LIN {X 0,Y 390.045,Z 635.903,A -85,B 0,C 180,E1 -11662.449,E2 -11662.449} C_VEL
LIN {X 0,Y 390.07,Z 635.897,A -85,B 0,C 180,E1 -11665.975,E2 -11665.975} C_VEL
LIN {X 0,Y 390.048,Z 635.899,A -85,B 0,C 180,E1 -11669.869,E2 -11669.869} C_VEL
LIN {X 0,Y 390.115,Z 635.892,A -85,B 0,C 180,E1 -11673.232,E2 -11673.232} C_VEL
LIN {X 0,Y 390.108,Z 635.894,A -85,B 0,C 180,E1 -11676.75,E2 -11676.75} C_VEL
LIN {X 0,Y 390.106,Z 635.893,A -85,B 0,C 180,E1 -11679.983,E2 -11679.983} C_VEL
LIN {X 0,Y 390.14,Z 635.89,A -85,B 0,C 180,E1 -11683.248,E2 -11683.248} C_VEL
LIN {X 0,Y 390.196,Z 635.883,A -85,B 0,C 180,E1 -11686.562,E2 -11686.562} C_VEL
LIN {X 0,Y 390.207,Z 635.88,A -85,B 0,C 180,E1 -11690.671,E2 -11690.671} C_VEL
LIN {X 0,Y 390.32,Z 635.867,A -85,B 0,C 180,E1 -11692.759,E2 -11692.759} C_VEL
LIN {X 0,Y 390.228,Z 635.88,A -85,B 0,C 180,E1 -11694.834,E2 -11694.834} C_VEL
LIN {X 0,Y 390.42,Z 635.855,A -85,B 0,C 180,E1 -11697.937,E2 -11697.937} C_VEL
LIN {X 0,Y 390.552,Z 635.838,A -85,B 0,C 180,E1 -11700,E2 -11700} C_VEL
LIN {X 0,Y 390.318,Z 635.869,A -85,B 0,C 180,E1 -11703.097,E2 -11703.097} C_VEL
LIN {X 0,Y 390.299,Z 635.869,A -85,B 0,C 180,E1 -11706.625,E2 -11706.625} C_VEL
LIN {X 0,Y 390.294,Z 635.871,A -85,B 0,C 180,E1 -11707.241,E2 -11707.241} C_VEL
LIN {X 0,Y 390.333,Z 637.799,A -85,B 0,C 180,E1 -11709.326,E2 -11709.326} C_VEL
LIN {X 0,Y 390.128,Z 641.266,A -85,B 0,C 180,E1 -11712.485,E2 -11712.485} C_VEL
LIN {X 0,Y 389.83,Z 644.908,A -85,B 0,C 180,E1 -11715.69,E2 -11715.69} C_VEL
LIN {X 0,Y 389.633,Z 648.746,A -85,B 0,C 180,E1 -11718.946,E2 -11718.946} C_VEL
LIN {X 0,Y 389.361,Z 652.799,A -85,B 0,C 180,E1 -11722.275,E2 -11722.275} C_VEL
LIN {X 0,Y 389.179,Z 657.06,A -85,B 0,C 180,E1 -11725.684,E2 -11725.684} C_VEL
LIN {X 0,Y 389.178,Z 658.085,A -85,B 0,C 180,E1 -11726.332,E2 -11726.332} C_VEL
LIN {X 0,Y 392.474,Z 670.829,A -85,B 0,C 180,E1 -11726.99,E2 -11726.99} C_VEL
LIN {X 0,Y 394.705,Z 682.309,A -85,B 0,C 180,E1 -11727.722,E2 -11727.722} C_VEL
LIN {X 0,Y 394.988,Z 685.201,A -85,B 0,C 180,E1 -11727.916,E2 -11727.916} C_VEL
LIN {X 0,Y 394.073,Z 697.293,A -85,B 0,C 180,E1 -11728.785,E2 -11728.785} C_VEL
LIN {X 0,Y 393.149,Z 709.316,A -85,B 0,C 180,E1 -11729.905,E2 -11729.905} C_VEL
LIN {X 0,Y 392.133,Z 719.9,A -85,B 0,C 180,E1 -11731.156,E2 -11731.156} C_VEL
LIN {X 0,Y 391.275,Z 729.716,A -85,B 0,C 180,E1 -11732.606,E2 -11732.606} C_VEL
LIN {X 0,Y 390.488,Z 737.933,A -85,B 0,C 180,E1 -11734.115,E2 -11734.115} C_VEL
LIN {X 0,Y 389.802,Z 745.117,A -85,B 0,C 180,E1 -11735.773,E2 -11735.773} C_VEL
LIN {X 0,Y 389.344,Z 750.732,A -85,B 0,C 180,E1 -11737.416,E2 -11737.416} C_VEL
LIN {X 0,Y 389,Z 755.433,A -85,B 0,C 180,E1 -11739.223,E2 -11739.223} C_VEL
LIN {X 0,Y 388.797,Z 758.049,A -85,B 0,C 180,E1 -11740.606,E2 -11740.606} C_VEL
LIN {X 0,Y 388.642,Z 760.083,A -85,B 0,C 180,E1 -11742.147,E2 -11742.147} C_VEL
LIN {X 0,Y 388.547,Z 761.204,A -85,B 0,C 180,E1 -11743.654,E2 -11743.654} C_VEL
LIN {X 0,Y 388.507,Z 761.496,A -85,B 0,C 180,E1 -11745.13,E2 -11745.13} C_VEL
LIN {X 0,Y 388.52,Z 761.002,A -85,B 0,C 180,E1 -11746.576,E2 -11746.576} C_VEL
LIN {X 0,Y 388.613,Z 759.717,A -85,B 0,C 180,E1 -11747.999,E2 -11747.999} C_VEL
LIN {X 0,Y 388.87,Z 756.445,A -85,B 0,C 180,E1 -11750.089,E2 -11750.089} C_VEL
LIN {X 0,Y 389.073,Z 753.106,A -85,B 0,C 180,E1 -11751.549,E2 -11751.549} C_VEL
LIN {X 0,Y 389.47,Z 747.243,A -85,B 0,C 180,E1 -11753.452,E2 -11753.452} C_VEL
LIN {X 0,Y 390.007,Z 740.747,A -85,B 0,C 180,E1 -11755.082,E2 -11755.082} C_VEL
LIN {X 0,Y 390.537,Z 734.245,A -85,B 0,C 180,E1 -11756.401,E2 -11756.401} C_VEL
LIN {X 0,Y 391.291,Z 725.804,A -85,B 0,C 180,E1 -11757.81,E2 -11757.81} C_VEL
LIN {X 0,Y 392.183,Z 715.296,A -85,B 0,C 180,E1 -11759.218,E2 -11759.218} C_VEL
LIN {X 0,Y 393.07,Z 704.453,A -85,B 0,C 180,E1 -11760.382,E2 -11760.382} C_VEL
LIN {X 0,Y 393.86,Z 693.01,A -85,B 0,C 180,E1 -11761.351,E2 -11761.351} C_VEL
LIN {X 0,Y 394.476,Z 683.755,A -85,B 0,C 180,E1 -11761.977,E2 -11761.977} C_VEL
LIN {X 0,Y 392.239,Z 671.38,A -85,B 0,C 180,E1 -11762.74,E2 -11762.74} C_VEL
LIN {X 0,Y 389.29,Z 658.629,A -85,B 0,C 180,E1 -11763.351,E2 -11763.351} C_VEL
LIN {X 0,Y 389.019,Z 657.042,A -85,B 0,C 180,E1 -11763.44,E2 -11763.44} C_VEL
LIN {X 0,Y 389.155,Z 652.247,A -85,B 0,C 180,E1 -11767.08,E2 -11767.08} C_VEL
LIN {X 0,Y 389.385,Z 648.528,A -85,B 0,C 180,E1 -11769.944,E2 -11769.944} C_VEL
LIN {X 0,Y 389.561,Z 644.36,A -85,B 0,C 180,E1 -11773.222,E2 -11773.222} C_VEL
LIN {X 0,Y 389.876,Z 639.95,A -85,B 0,C 180,E1 -11776.76,E2 -11776.76} C_VEL
LIN {X 0,Y 389.963,Z 636.512,A -85,B 0,C 180,E1 -11779.617,E2 -11779.617} C_VEL
LIN {X 0,Y 390.071,Z 635.898,A -85,B 0,C 180,E1 -11780.668,E2 -11780.668} C_VEL
LIN {X 0,Y 390.293,Z 635.871,A -85,B 0,C 180,E1 -11782.758,E2 -11782.758} C_VEL
LIN {X 0,Y 390.229,Z 635.879,A -85,B 0,C 180,E1 -11784.833,E2 -11784.833} C_VEL
LIN {X 0,Y 390.424,Z 635.849,A -85,B 0,C 180,E1 -11787.936,E2 -11787.936} C_VEL
LIN {X 0,Y 390.554,Z 635.834,A -85,B 0,C 180,E1 -11790,E2 -11790} C_VEL
LIN {X 0,Y 390.318,Z 635.867,A -85,B 0,C 180,E1 -11793.096,E2 -11793.096} C_VEL
LIN {X 0,Y 390.313,Z 635.864,A -85,B 0,C 180,E1 -11796.202,E2 -11796.202} C_VEL
LIN {X 0,Y 390.171,Z 635.883,A -85,B 0,C 180,E1 -11798.285,E2 -11798.285} C_VEL
LIN {X 0,Y 389.679,Z 635.945,A -85,B 0,C 180,E1 -11801.442,E2 -11801.442} C_VEL
LIN {X 0,Y 389.557,Z 636.18,A -85,B 0,C 180,E1 -11802.238,E2 -11802.238} C_VEL
LIN {X 0,Y 389.338,Z 640.085,A -85,B 0,C 180,E1 -11804.837,E2 -11804.837} C_VEL
LIN {X 0,Y 388.609,Z 641.43,A -85,B 0,C 180,E1 -11805.677,E2 -11805.677} C_VEL
LIN {X 0,Y 385.67,Z 643.774,A -85,B 0,C 180,E1 -11807.034,E2 -11807.034} C_VEL
LIN {X 0,Y 383.212,Z 645.663,A -85,B 0,C 180,E1 -11808.131,E2 -11808.131} C_VEL
LIN {X 0,Y 382.164,Z 647.033,A -85,B 0,C 180,E1 -11808.983,E2 -11808.983} C_VEL
LIN {X 0,Y 382.081,Z 647.468,A -85,B 0,C 180,E1 -11809.272,E2 -11809.272} C_VEL
LIN {X 0,Y 381.91,Z 653.113,A -85,B 0,C 180,E1 -11813.057,E2 -11813.057} C_VEL
LIN {X 0,Y 381.878,Z 656.667,A -85,B 0,C 180,E1 -11815.387,E2 -11815.387} C_VEL
LIN {X 0,Y 384.96,Z 670.347,A -85,B 0,C 180,E1 -11816.022,E2 -11816.022} C_VEL
LIN {X 0,Y 387.385,Z 683.195,A -85,B 0,C 180,E1 -11816.826,E2 -11816.826} C_VEL
LIN {X 0,Y 386.877,Z 694.197,A -85,B 0,C 180,E1 -11817.595,E2 -11817.595} C_VEL
LIN {X 0,Y 385.998,Z 705.968,A -85,B 0,C 180,E1 -11818.634,E2 -11818.634} C_VEL
LIN {X 0,Y 385.071,Z 716.555,A -85,B 0,C 180,E1 -11819.824,E2 -11819.824} C_VEL
LIN {X 0,Y 384.168,Z 726.914,A -85,B 0,C 180,E1 -11821.271,E2 -11821.271} C_VEL
LIN {X 0,Y 383.482,Z 734.296,A -85,B 0,C 180,E1 -11822.538,E2 -11822.538} C_VEL
LIN {X 0,Y 382.975,Z 740.583,A -85,B 0,C 180,E1 -11823.836,E2 -11823.836} C_VEL
LIN {X 0,Y 382.455,Z 746.653,A -85,B 0,C 180,E1 -11825.356,E2 -11825.356} C_VEL
LIN {X 0,Y 382.09,Z 751.026,A -85,B 0,C 180,E1 -11826.711,E2 -11826.711} C_VEL
LIN {X 0,Y 381.844,Z 754.811,A -85,B 0,C 180,E1 -11828.181,E2 -11828.181} C_VEL
LIN {X 0,Y 381.522,Z 758.493,A -85,B 0,C 180,E1 -11830.145,E2 -11830.145} C_VEL
LIN {X 0,Y 381.417,Z 760.21,A -85,B 0,C 180,E1 -11831.554,E2 -11831.554} C_VEL
LIN {X 0,Y 381.35,Z 761.195,A -85,B 0,C 180,E1 -11832.99,E2 -11832.99} C_VEL
LIN {X 0,Y 381.403,Z 761.452,A -85,B 0,C 180,E1 -11834.443,E2 -11834.443} C_VEL
LIN {X 0,Y 381.435,Z 760.939,A -85,B 0,C 180,E1 -11835.936,E2 -11835.936} C_VEL
LIN {X 0,Y 381.547,Z 759.581,A -85,B 0,C 180,E1 -11837.458,E2 -11837.458} C_VEL
LIN {X 0,Y 381.702,Z 757.288,A -85,B 0,C 180,E1 -11839.016,E2 -11839.016} C_VEL
LIN {X 0,Y 382.005,Z 753.991,A -85,B 0,C 180,E1 -11840.596,E2 -11840.596} C_VEL
LIN {X 0,Y 382.384,Z 749.518,A -85,B 0,C 180,E1 -11842.214,E2 -11842.214} C_VEL
LIN {X 0,Y 382.967,Z 742.914,A -85,B 0,C 180,E1 -11844.038,E2 -11844.038} C_VEL
LIN {X 0,Y 383.596,Z 736.113,A -85,B 0,C 180,E1 -11845.533,E2 -11845.533} C_VEL
LIN {X 0,Y 384.492,Z 727.815,A -85,B 0,C 180,E1 -11847.013,E2 -11847.013} C_VEL
LIN {X 0,Y 385.344,Z 719.065,A -85,B 0,C 180,E1 -11848.285,E2 -11848.285} C_VEL
LIN {X 0,Y 386.37,Z 708.31,A -85,B 0,C 180,E1 -11849.548,E2 -11849.548} C_VEL
LIN {X 0,Y 387.261,Z 697.305,A -85,B 0,C 180,E1 -11850.586,E2 -11850.586} C_VEL
LIN {X 0,Y 388.115,Z 685.408,A -85,B 0,C 180,E1 -11851.453,E2 -11851.453} C_VEL
LIN {X 0,Y 386.153,Z 673.731,A -85,B 0,C 180,E1 -11852.242,E2 -11852.242} C_VEL
LIN {X 0,Y 383.142,Z 661.505,A -85,B 0,C 180,E1 -11852.926,E2 -11852.926} C_VEL
LIN {X 0,Y 381.987,Z 657.119,A -85,B 0,C 180,E1 -11853.133,E2 -11853.133} C_VEL
LIN {X 0,Y 382.071,Z 652.636,A -85,B 0,C 180,E1 -11856.129,E2 -11856.129} C_VEL
LIN {X 0,Y 382.223,Z 647.235,A -85,B 0,C 180,E1 -11859.674,E2 -11859.674} C_VEL
LIN {X 0,Y 382.36,Z 642.32,A -85,B 0,C 180,E1 -11862.897,E2 -11862.897} C_VEL
LIN {X 0,Y 382.677,Z 636.826,A -85,B 0,C 180,E1 -11866.478,E2 -11866.478} C_VEL
LIN {X 0,Y 383.006,Z 636.779,A -85,B 0,C 180,E1 -11869.426,E2 -11869.426} C_VEL
LIN {X 0,Y 383.25,Z 636.75,A -85,B 0,C 180,E1 -11872.625,E2 -11872.625} C_VEL
LIN {X 0,Y 383.196,Z 636.756,A -85,B 0,C 180,E1 -11874.738,E2 -11874.738} C_VEL
LIN {X 0,Y 383.385,Z 636.731,A -85,B 0,C 180,E1 -11877.899,E2 -11877.899} C_VEL
LIN {X 0,Y 383.518,Z 636.715,A -85,B 0,C 180,E1 -11880,E2 -11880} C_VEL
LIN {X 0,Y 383.249,Z 636.749,A -85,B 0,C 180,E1 -11883.154,E2 -11883.154} C_VEL
LIN {X 0,Y 383.284,Z 636.743,A -85,B 0,C 180,E1 -11886.316,E2 -11886.316} C_VEL
LIN {X 0,Y 383.256,Z 636.747,A -85,B 0,C 180,E1 -11888.436,E2 -11888.436} C_VEL
LIN {X 0,Y 383.095,Z 636.766,A -85,B 0,C 180,E1 -11891.642,E2 -11891.642} C_VEL
LIN {X 0,Y 383.106,Z 636.766,A -85,B 0,C 180,E1 -11894.882,E2 -11894.882} C_VEL
LIN {X 0,Y 383.085,Z 636.768,A -85,B 0,C 180,E1 -11898.172,E2 -11898.172} C_VEL
LIN {X 0,Y 382.989,Z 636.777,A -85,B 0,C 180,E1 -11901.531,E2 -11901.531} C_VEL
LIN {X 0,Y 383.049,Z 636.773,A -85,B 0,C 180,E1 -11904.961,E2 -11904.961} C_VEL
LIN {X 0,Y 383.046,Z 636.77,A -85,B 0,C 180,E1 -11908.492,E2 -11908.492} C_VEL
LIN {X 0,Y 383.008,Z 636.779,A -85,B 0,C 180,E1 -11912.15,E2 -11912.15} C_VEL
LIN {X 0,Y 383.015,Z 636.776,A -85,B 0,C 180,E1 -11914.668,E2 -11914.668} C_VEL
LIN {X 0,Y 382.999,Z 636.777,A -85,B 0,C 180,E1 -11917.905,E2 -11917.905} C_VEL
LIN {X 0,Y 382.981,Z 636.781,A -85,B 0,C 180,E1 -11921.348,E2 -11921.348} C_VEL
LIN {X 0,Y 382.993,Z 636.78,A -85,B 0,C 180,E1 -11924.304,E2 -11924.304} C_VEL
LIN {X 0,Y 383.029,Z 636.776,A -85,B 0,C 180,E1 -11928.132,E2 -11928.132} C_VEL
LIN {X 0,Y 383.63,Z 640,A -85,B 0,C 180,E1 -11930.303,E2 -11930.303} C_VEL
LIN {X 0,Y 384.197,Z 644.117,A -85,B 0,C 180,E1 -11932.868,E2 -11932.868} C_VEL
LIN {X 0,Y 384.255,Z 648.497,A -85,B 0,C 180,E1 -11935.46,E2 -11935.46} C_VEL
LIN {X 0,Y 383.782,Z 653.949,A -85,B 0,C 180,E1 -11938.541,E2 -11938.541} C_VEL
LIN {X 0,Y 383.349,Z 659.601,A -85,B 0,C 180,E1 -11941.642,E2 -11941.642} C_VEL
LIN {X 0,Y 382.888,Z 665.937,A -85,B 0,C 180,E1 -11945.029,E2 -11945.029} C_VEL
LIN {X 0,Y 382.537,Z 672.453,A -85,B 0,C 180,E1 -11948.443,E2 -11948.443} C_VEL
LIN {X 0,Y 382.233,Z 677.92,A -85,B 0,C 180,E1 -11951.214,E2 -11951.214} C_VEL
LIN {X 0,Y 384.658,Z 691.057,A -85,B 0,C 180,E1 -11951.82,E2 -11951.82} C_VEL
LIN {X 0,Y 386.51,Z 704.837,A -85,B 0,C 180,E1 -11952.638,E2 -11952.638} C_VEL
LIN {X 0,Y 387.056,Z 710.39,A -85,B 0,C 180,E1 -11953.022,E2 -11953.022} C_VEL
LIN {X 0,Y 386.176,Z 721.714,A -85,B 0,C 180,E1 -11953.887,E2 -11953.887} C_VEL
LIN {X 0,Y 385.325,Z 732.5,A -85,B 0,C 180,E1 -11954.936,E2 -11954.936} C_VEL
LIN {X 0,Y 384.394,Z 743.32,A -85,B 0,C 180,E1 -11956.251,E2 -11956.251} C_VEL
LIN {X 0,Y 383.627,Z 752.108,A -85,B 0,C 180,E1 -11957.57,E2 -11957.57} C_VEL
LIN {X 0,Y 382.854,Z 760.667,A -85,B 0,C 180,E1 -11959.155,E2 -11959.155} C_VEL
LIN {X 0,Y 382.309,Z 767.528,A -85,B 0,C 180,E1 -11960.744,E2 -11960.744} C_VEL
LIN {X 0,Y 381.868,Z 773.826,A -85,B 0,C 180,E1 -11962.599,E2 -11962.599} C_VEL
LIN {X 0,Y 381.697,Z 777.168,A -85,B 0,C 180,E1 -11963.868,E2 -11963.868} C_VEL
LIN {X 0,Y 381.633,Z 780.953,A -85,B 0,C 180,E1 -11965.776,E2 -11965.776} C_VEL
LIN {X 0,Y 381.545,Z 782.431,A -85,B 0,C 180,E1 -11966.833,E2 -11966.833} C_VEL
LIN {X 0,Y 381.616,Z 784.105,A -85,B 0,C 180,E1 -11968.945,E2 -11968.945} C_VEL
LIN {X 0,Y 381.639,Z 784.353,A -85,B 0,C 180,E1 -11970,E2 -11970} C_VEL
LIN {X 0,Y 381.616,Z 784.185,A -85,B 0,C 180,E1 -11971.056,E2 -11971.056} C_VEL
LIN {X 0,Y 381.544,Z 782.599,A -85,B 0,C 180,E1 -11973.168,E2 -11973.168} C_VEL
LIN {X 0,Y 381.634,Z 781.213,A -85,B 0,C 180,E1 -11974.225,E2 -11974.225} C_VEL
LIN {X 0,Y 381.734,Z 777.457,A -85,B 0,C 180,E1 -11976.184,E2 -11976.184} C_VEL
LIN {X 0,Y 382.012,Z 772.753,A -85,B 0,C 180,E1 -11977.931,E2 -11977.931} C_VEL
LIN {X 0,Y 382.498,Z 766.218,A -85,B 0,C 180,E1 -11979.786,E2 -11979.786} C_VEL
LIN {X 0,Y 383.092,Z 759.074,A -85,B 0,C 180,E1 -11981.374,E2 -11981.374} C_VEL
LIN {X 0,Y 384.032,Z 750.186,A -85,B 0,C 180,E1 -11982.955,E2 -11982.955} C_VEL
LIN {X 0,Y 384.832,Z 740.922,A -85,B 0,C 180,E1 -11984.299,E2 -11984.299} C_VEL
LIN {X 0,Y 385.707,Z 731.154,A -85,B 0,C 180,E1 -11985.455,E2 -11985.455} C_VEL
LIN {X 0,Y 386.704,Z 720.176,A -85,B 0,C 180,E1 -11986.498,E2 -11986.498} C_VEL
LIN {X 0,Y 387.423,Z 709.101,A -85,B 0,C 180,E1 -11987.34,E2 -11987.34} C_VEL
LIN {X 0,Y 386.021,Z 696.528,A -85,B 0,C 180,E1 -11988.181,E2 -11988.181} C_VEL
LIN {X 0,Y 383.884,Z 684.526,A -85,B 0,C 180,E1 -11988.827,E2 -11988.827} C_VEL
LIN {X 0,Y 382.267,Z 677.169,A -85,B 0,C 180,E1 -11989.162,E2 -11989.162} C_VEL
LIN {X 0,Y 382.62,Z 671.462,A -85,B 0,C 180,E1 -11992.12,E2 -11992.12} C_VEL
LIN {X 0,Y 383.018,Z 664.285,A -85,B 0,C 180,E1 -11995.959,E2 -11995.959} C_VEL
LIN {X 0,Y 383.468,Z 658.701,A -85,B 0,C 180,E1 -11999.057,E2 -11999.057} C_VEL
LIN {X 0,Y 384.047,Z 652.474,A -85,B 0,C 180,E1 -12002.67,E2 -12002.67} C_VEL
LIN {X 0,Y 384.393,Z 649.227,A -85,B 0,C 180,E1 -12004.639,E2 -12004.639} C_VEL
LIN {X 0,Y 384.313,Z 645.402,A -85,B 0,C 180,E1 -12007.12,E2 -12007.12} C_VEL
LIN {X 0,Y 383.808,Z 641.495,A -85,B 0,C 180,E1 -12009.859,E2 -12009.859} C_VEL
LIN {X 0,Y 383.035,Z 636.776,A -85,B 0,C 180,E1 -12013.567,E2 -12013.567} C_VEL
LIN {X 0,Y 383.012,Z 636.78,A -85,B 0,C 180,E1 -12017.24,E2 -12017.24} C_VEL
LIN {X 0,Y 383.017,Z 636.778,A -85,B 0,C 180,E1 -12020.414,E2 -12020.414} C_VEL
LIN {X 0,Y 383.027,Z 636.776,A -85,B 0,C 180,E1 -12024.045,E2 -12024.045} C_VEL
LIN {X 0,Y 382.988,Z 636.779,A -85,B 0,C 180,E1 -12027.578,E2 -12027.578} C_VEL
LIN {X 0,Y 382.994,Z 636.779,A -85,B 0,C 180,E1 -12030.3,E2 -12030.3} C_VEL
LIN {X 0,Y 383.082,Z 636.766,A -85,B 0,C 180,E1 -12034.021,E2 -12034.021} C_VEL
LIN {X 0,Y 383.01,Z 636.778,A -85,B 0,C 180,E1 -12037.335,E2 -12037.335} C_VEL
LIN {X 0,Y 383.062,Z 636.772,A -85,B 0,C 180,E1 -12040.716,E2 -12040.716} C_VEL
LIN {X 0,Y 383.082,Z 636.768,A -85,B 0,C 180,E1 -12044.027,E2 -12044.027} C_VEL
LIN {X 0,Y 383.138,Z 636.761,A -85,B 0,C 180,E1 -12047.284,E2 -12047.284} C_VEL
LIN {X 0,Y 383.153,Z 636.758,A -85,B 0,C 180,E1 -12050.498,E2 -12050.498} C_VEL
LIN {X 0,Y 383.275,Z 636.743,A -85,B 0,C 180,E1 -12052.625,E2 -12052.625} C_VEL
LIN {X 0,Y 383.201,Z 636.754,A -85,B 0,C 180,E1 -12054.739,E2 -12054.739} C_VEL
LIN {X 0,Y 383.387,Z 636.731,A -85,B 0,C 180,E1 -12057.899,E2 -12057.899} C_VEL
LIN {X 0,Y 383.521,Z 636.714,A -85,B 0,C 180,E1 -12060,E2 -12060} C_VEL
LIN {X 0,Y 383.254,Z 636.75,A -85,B 0,C 180,E1 -12063.154,E2 -12063.154} C_VEL
LIN {X 0,Y 383.271,Z 636.803,A -85,B 0,C 180,E1 -12066.622,E2 -12066.622} C_VEL
LIN {X 0,Y 383.287,Z 636.949,A -85,B 0,C 180,E1 -12067.374,E2 -12067.374} C_VEL
LIN {X 0,Y 383.241,Z 640.208,A -85,B 0,C 180,E1 -12070.567,E2 -12070.567} C_VEL
LIN {X 0,Y 382.991,Z 643.756,A -85,B 0,C 180,E1 -12073.801,E2 -12073.801} C_VEL
LIN {X 0,Y 382.689,Z 647.682,A -85,B 0,C 180,E1 -12077.26,E2 -12077.26} C_VEL
LIN {X 0,Y 382.449,Z 651.413,A -85,B 0,C 180,E1 -12080.435,E2 -12080.435} C_VEL
LIN {X 0,Y 382.211,Z 655.568,A -85,B 0,C 180,E1 -12083.862,E2 -12083.862} C_VEL
LIN {X 0,Y 382.103,Z 658.125,A -85,B 0,C 180,E1 -12085.928,E2 -12085.928} C_VEL
LIN {X 0,Y 385.596,Z 671.291,A -85,B 0,C 180,E1 -12086.631,E2 -12086.631} C_VEL
LIN {X 0,Y 387.809,Z 682.676,A -85,B 0,C 180,E1 -12087.377,E2 -12087.377} C_VEL
LIN {X 0,Y 388.111,Z 687.57,A -85,B 0,C 180,E1 -12087.72,E2 -12087.72} C_VEL
LIN {X 0,Y 387.174,Z 699.209,A -85,B 0,C 180,E1 -12088.605,E2 -12088.605} C_VEL
LIN {X 0,Y 386.243,Z 710.637,A -85,B 0,C 180,E1 -12089.725,E2 -12089.725} C_VEL
LIN {X 0,Y 385.225,Z 720.768,A -85,B 0,C 180,E1 -12090.967,E2 -12090.967} C_VEL
LIN {X 0,Y 384.345,Z 729.91,A -85,B 0,C 180,E1 -12092.35,E2 -12092.35} C_VEL
LIN {X 0,Y 383.538,Z 737.997,A -85,B 0,C 180,E1 -12093.858,E2 -12093.858} C_VEL
LIN {X 0,Y 382.779,Z 745.636,A -85,B 0,C 180,E1 -12095.658,E2 -12095.658} C_VEL
LIN {X 0,Y 382.277,Z 751.252,A -85,B 0,C 180,E1 -12097.351,E2 -12097.351} C_VEL
LIN {X 0,Y 381.998,Z 754.801,A -85,B 0,C 180,E1 -12098.721,E2 -12098.721} C_VEL
LIN {X 0,Y 381.785,Z 757.62,A -85,B 0,C 180,E1 -12100.113,E2 -12100.113} C_VEL
LIN {X 0,Y 381.582,Z 759.732,A -85,B 0,C 180,E1 -12101.533,E2 -12101.533} C_VEL
LIN {X 0,Y 381.502,Z 761.063,A -85,B 0,C 180,E1 -12102.97,E2 -12102.97} C_VEL
LIN {X 0,Y 381.421,Z 761.675,A -85,B 0,C 180,E1 -12104.442,E2 -12104.442} C_VEL
LIN {X 0,Y 381.412,Z 761.516,A -85,B 0,C 180,E1 -12105.941,E2 -12105.941} C_VEL
LIN {X 0,Y 381.468,Z 760.524,A -85,B 0,C 180,E1 -12107.472,E2 -12107.472} C_VEL
LIN {X 0,Y 381.637,Z 758.614,A -85,B 0,C 180,E1 -12109.029,E2 -12109.029} C_VEL
LIN {X 0,Y 381.853,Z 755.698,A -85,B 0,C 180,E1 -12110.625,E2 -12110.625} C_VEL
LIN {X 0,Y 382.095,Z 751.605,A -85,B 0,C 180,E1 -12112.271,E2 -12112.271} C_VEL
LIN {X 0,Y 382.574,Z 745.965,A -85,B 0,C 180,E1 -12113.995,E2 -12113.995} C_VEL
LIN {X 0,Y 383.121,Z 739.116,A -85,B 0,C 180,E1 -12115.638,E2 -12115.638} C_VEL
LIN {X 0,Y 383.792,Z 731.872,A -85,B 0,C 180,E1 -12117.045,E2 -12117.045} C_VEL
LIN {X 0,Y 384.653,Z 722.225,A -85,B 0,C 180,E1 -12118.57,E2 -12118.57} C_VEL
LIN {X 0,Y 385.647,Z 711.389,A -85,B 0,C 180,E1 -12119.923,E2 -12119.923} C_VEL
LIN {X 0,Y 386.502,Z 700.447,A -85,B 0,C 180,E1 -12121.02,E2 -12121.02} C_VEL
LIN {X 0,Y 387.303,Z 689.022,A -85,B 0,C 180,E1 -12121.922,E2 -12121.922} C_VEL
LIN {X 0,Y 387.451,Z 683.305,A -85,B 0,C 180,E1 -12122.302,E2 -12122.302} C_VEL
LIN {X 0,Y 384.754,Z 669.527,A -85,B 0,C 180,E1 -12123.159,E2 -12123.159} C_VEL
LIN {X 0,Y 382.003,Z 657.244,A -85,B 0,C 180,E1 -12123.76,E2 -12123.76} C_VEL
LIN {X 0,Y 382.105,Z 652.674,A -85,B 0,C 180,E1 -12127.278,E2 -12127.278} C_VEL
LIN {X 0,Y 382.332,Z 648.341,A -85,B 0,C 180,E1 -12130.678,E2 -12130.678} C_VEL
LIN {X 0,Y 382.533,Z 644.196,A -85,B 0,C 180,E1 -12134.003,E2 -12134.003} C_VEL
LIN {X 0,Y 382.858,Z 640.183,A -85,B 0,C 180,E1 -12137.274,E2 -12137.274} C_VEL
LIN {X 0,Y 382.895,Z 637.635,A -85,B 0,C 180,E1 -12139.423,E2 -12139.423} C_VEL
LIN {X 0,Y 382.996,Z 636.779,A -85,B 0,C 180,E1 -12140.494,E2 -12140.494} C_VEL
LIN {X 0,Y 383.242,Z 636.747,A -85,B 0,C 180,E1 -12142.624,E2 -12142.624} C_VEL
LIN {X 0,Y 383.201,Z 636.754,A -85,B 0,C 180,E1 -12144.738,E2 -12144.738} C_VEL
LIN {X 0,Y 383.391,Z 636.725,A -85,B 0,C 180,E1 -12147.899,E2 -12147.899} C_VEL
LIN {X 0,Y 383.523,Z 636.709,A -85,B 0,C 180,E1 -12150,E2 -12150} C_VEL
LIN {X 0,Y 383.254,Z 636.746,A -85,B 0,C 180,E1 -12153.153,E2 -12153.153} C_VEL
LIN {X 0,Y 383.265,Z 636.743,A -85,B 0,C 180,E1 -12156.316,E2 -12156.316} C_VEL
LIN {X 0,Y 383.106,Z 636.764,A -85,B 0,C 180,E1 -12158.439,E2 -12158.439} C_VEL
LIN {X 0,Y 382.547,Z 636.833,A -85,B 0,C 180,E1 -12162.096,E2 -12162.096} C_VEL
LIN {X 0,Y 382.258,Z 642.612,A -85,B 0,C 180,E1 -12166.008,E2 -12166.008} C_VEL
LIN {X 0,Y 382.081,Z 647.468,A -85,B 0,C 180,E1 -12169.272,E2 -12169.272} C_VEL
LIN {X 0,Y 381.403,Z 648.808,A -85,B 0,C 180,E1 -12170.128,E2 -12170.128} C_VEL
LIN {X 0,Y 378.476,Z 651.152,A -85,B 0,C 180,E1 -12171.512,E2 -12171.512} C_VEL
LIN {X 0,Y 375.98,Z 653.04,A -85,B 0,C 180,E1 -12172.63,E2 -12172.63} C_VEL
LIN {X 0,Y 374.892,Z 654.419,A -85,B 0,C 180,E1 -12173.498,E2 -12173.498} C_VEL
LIN {X 0,Y 374.795,Z 654.862,A -85,B 0,C 180,E1 -12173.793,E2 -12173.793} C_VEL
LIN {X 0,Y 374.785,Z 656.69,A -85,B 0,C 180,E1 -12175.029,E2 -12175.029} C_VEL
LIN {X 0,Y 378.148,Z 671.675,A -85,B 0,C 180,E1 -12175.772,E2 -12175.772} C_VEL
LIN {X 0,Y 380.536,Z 684.409,A -85,B 0,C 180,E1 -12176.606,E2 -12176.606} C_VEL
LIN {X 0,Y 379.958,Z 695.309,A -85,B 0,C 180,E1 -12177.396,E2 -12177.396} C_VEL
LIN {X 0,Y 379.119,Z 705.958,A -85,B 0,C 180,E1 -12178.361,E2 -12178.361} C_VEL
LIN {X 0,Y 378.204,Z 716.023,A -85,B 0,C 180,E1 -12179.498,E2 -12179.498} C_VEL
LIN {X 0,Y 377.388,Z 725.09,A -85,B 0,C 180,E1 -12180.755,E2 -12180.755} C_VEL
LIN {X 0,Y 376.612,Z 733.265,A -85,B 0,C 180,E1 -12182.129,E2 -12182.129} C_VEL
LIN {X 0,Y 375.907,Z 741.288,A -85,B 0,C 180,E1 -12183.793,E2 -12183.793} C_VEL
LIN {X 0,Y 375.345,Z 747.708,A -85,B 0,C 180,E1 -12185.481,E2 -12185.481} C_VEL
LIN {X 0,Y 374.849,Z 753.478,A -85,B 0,C 180,E1 -12187.445,E2 -12187.445} C_VEL
LIN {X 0,Y 374.604,Z 756.736,A -85,B 0,C 180,E1 -12188.938,E2 -12188.938} C_VEL
LIN {X 0,Y 374.353,Z 759.926,A -85,B 0,C 180,E1 -12191.077,E2 -12191.077} C_VEL
LIN {X 0,Y 374.252,Z 761.354,A -85,B 0,C 180,E1 -12192.914,E2 -12192.914} C_VEL
LIN {X 0,Y 374.306,Z 761.65,A -85,B 0,C 180,E1 -12194.48,E2 -12194.48} C_VEL
LIN {X 0,Y 374.341,Z 761.137,A -85,B 0,C 180,E1 -12196,E2 -12196} C_VEL
LIN {X 0,Y 374.455,Z 759.84,A -85,B 0,C 180,E1 -12197.494,E2 -12197.494} C_VEL
LIN {X 0,Y 374.612,Z 757.777,A -85,B 0,C 180,E1 -12198.957,E2 -12198.957} C_VEL
LIN {X 0,Y 374.879,Z 754.965,A -85,B 0,C 180,E1 -12200.401,E2 -12200.401} C_VEL
LIN {X 0,Y 375.298,Z 750.255,A -85,B 0,C 180,E1 -12202.21,E2 -12202.21} C_VEL
LIN {X 0,Y 375.694,Z 745.808,A -85,B 0,C 180,E1 -12203.55,E2 -12203.55} C_VEL
LIN {X 0,Y 376.409,Z 738.896,A -85,B 0,C 180,E1 -12205.237,E2 -12205.237} C_VEL
LIN {X 0,Y 377.249,Z 731.108,A -85,B 0,C 180,E1 -12206.761,E2 -12206.761} C_VEL
LIN {X 0,Y 378.217,Z 722.13,A -85,B 0,C 180,E1 -12208.18,E2 -12208.18} C_VEL
LIN {X 0,Y 379.267,Z 711.683,A -85,B 0,C 180,E1 -12209.518,E2 -12209.518} C_VEL
LIN {X 0,Y 380.299,Z 700.109,A -85,B 0,C 180,E1 -12210.688,E2 -12210.688} C_VEL
LIN {X 0,Y 381.319,Z 687.632,A -85,B 0,C 180,E1 -12211.667,E2 -12211.667} C_VEL
LIN {X 0,Y 380.77,Z 682.073,A -85,B 0,C 180,E1 -12212.072,E2 -12212.072} C_VEL
LIN {X 0,Y 378.115,Z 669.238,A -85,B 0,C 180,E1 -12212.91,E2 -12212.91} C_VEL
LIN {X 0,Y 374.951,Z 657.3,A -85,B 0,C 180,E1 -12213.555,E2 -12213.555} C_VEL
LIN {X 0,Y 375.033,Z 652.43,A -85,B 0,C 180,E1 -12216.825,E2 -12216.825} C_VEL
LIN {X 0,Y 375.19,Z 647.219,A -85,B 0,C 180,E1 -12220.295,E2 -12220.295} C_VEL
LIN {X 0,Y 375.341,Z 642.042,A -85,B 0,C 180,E1 -12223.688,E2 -12223.688} C_VEL
LIN {X 0,Y 375.656,Z 637.701,A -85,B 0,C 180,E1 -12226.614,E2 -12226.614} C_VEL
LIN {X 0,Y 376.041,Z 637.646,A -85,B 0,C 180,E1 -12230.316,E2 -12230.316} C_VEL
LIN {X 0,Y 376.204,Z 637.628,A -85,B 0,C 180,E1 -12232.486,E2 -12232.486} C_VEL
LIN {X 0,Y 376.168,Z 637.631,A -85,B 0,C 180,E1 -12234.64,E2 -12234.64} C_VEL
LIN {X 0,Y 376.351,Z 637.607,A -85,B 0,C 180,E1 -12237.86,E2 -12237.86} C_VEL
LIN {X 0,Y 376.487,Z 637.591,A -85,B 0,C 180,E1 -12240,E2 -12240} C_VEL
LIN {X 0,Y 376.187,Z 637.629,A -85,B 0,C 180,E1 -12243.213,E2 -12243.213} C_VEL
LIN {X 0,Y 376.243,Z 637.621,A -85,B 0,C 180,E1 -12246.435,E2 -12246.435} C_VEL
LIN {X 0,Y 376.201,Z 637.627,A -85,B 0,C 180,E1 -12248.595,E2 -12248.595} C_VEL
LIN {X 0,Y 376.047,Z 637.643,A -85,B 0,C 180,E1 -12251.864,E2 -12251.864} C_VEL
LIN {X 0,Y 376.054,Z 637.644,A -85,B 0,C 180,E1 -12255.168,E2 -12255.168} C_VEL
LIN {X 0,Y 376.02,Z 637.648,A -85,B 0,C 180,E1 -12258.526,E2 -12258.526} C_VEL
LIN {X 0,Y 375.96,Z 637.655,A -85,B 0,C 180,E1 -12261.955,E2 -12261.955} C_VEL
LIN {X 0,Y 376.003,Z 637.65,A -85,B 0,C 180,E1 -12265.461,E2 -12265.461} C_VEL
LIN {X 0,Y 375.973,Z 637.653,A -85,B 0,C 180,E1 -12269.079,E2 -12269.079} C_VEL
LIN {X 0,Y 375.946,Z 637.656,A -85,B 0,C 180,E1 -12272.829,E2 -12272.829} C_VEL
LIN {X 0,Y 375.955,Z 637.654,A -85,B 0,C 180,E1 -12275.416,E2 -12275.416} C_VEL
LIN {X 0,Y 375.973,Z 637.653,A -85,B 0,C 180,E1 -12278.271,E2 -12278.271} C_VEL
LIN {X 0,Y 375.932,Z 637.658,A -85,B 0,C 180,E1 -12281.601,E2 -12281.601} C_VEL
LIN {X 0,Y 375.925,Z 637.661,A -85,B 0,C 180,E1 -12285.269,E2 -12285.269} C_VEL
LIN {X 0,Y 376.008,Z 637.835,A -85,B 0,C 180,E1 -12288.09,E2 -12288.09} C_VEL
LIN {X 0,Y 376.705,Z 641.685,A -85,B 0,C 180,E1 -12290.631,E2 -12290.631} C_VEL
LIN {X 0,Y 377.244,Z 646.098,A -85,B 0,C 180,E1 -12293.406,E2 -12293.406} C_VEL
LIN {X 0,Y 377.291,Z 648.82,A -85,B 0,C 180,E1 -12295.046,E2 -12295.046} C_VEL
LIN {X 0,Y 376.833,Z 653.729,A -85,B 0,C 180,E1 -12297.892,E2 -12297.892} C_VEL
LIN {X 0,Y 376.328,Z 659.921,A -85,B 0,C 180,E1 -12301.371,E2 -12301.371} C_VEL
LIN {X 0,Y 375.808,Z 666.787,A -85,B 0,C 180,E1 -12305.117,E2 -12305.117} C_VEL
LIN {X 0,Y 375.433,Z 673.303,A -85,B 0,C 180,E1 -12308.591,E2 -12308.591} C_VEL
LIN {X 0,Y 375.204,Z 677.515,A -85,B 0,C 180,E1 -12310.795,E2 -12310.795} C_VEL
LIN {X 0,Y 377.752,Z 690.907,A -85,B 0,C 180,E1 -12311.436,E2 -12311.436} C_VEL
LIN {X 0,Y 379.386,Z 702.934,A -85,B 0,C 180,E1 -12312.185,E2 -12312.185} C_VEL
LIN {X 0,Y 380.151,Z 711.124,A -85,B 0,C 180,E1 -12312.795,E2 -12312.795} C_VEL
LIN {X 0,Y 379.083,Z 724.101,A -85,B 0,C 180,E1 -12313.854,E2 -12313.854} C_VEL
LIN {X 0,Y 378.105,Z 735.658,A -85,B 0,C 180,E1 -12315.067,E2 -12315.067} C_VEL
LIN {X 0,Y 377.276,Z 744.815,A -85,B 0,C 180,E1 -12316.261,E2 -12316.261} C_VEL
LIN {X 0,Y 376.504,Z 753.282,A -85,B 0,C 180,E1 -12317.605,E2 -12317.605} C_VEL
LIN {X 0,Y 375.717,Z 761.552,A -85,B 0,C 180,E1 -12319.22,E2 -12319.22} C_VEL
LIN {X 0,Y 375.212,Z 768.218,A -85,B 0,C 180,E1 -12320.839,E2 -12320.839} C_VEL
LIN {X 0,Y 374.802,Z 773.524,A -85,B 0,C 180,E1 -12322.458,E2 -12322.458} C_VEL
LIN {X 0,Y 374.593,Z 777.276,A -85,B 0,C 180,E1 -12323.919,E2 -12323.919} C_VEL
LIN {X 0,Y 374.559,Z 780.694,A -85,B 0,C 180,E1 -12325.696,E2 -12325.696} C_VEL
LIN {X 0,Y 374.461,Z 782.189,A -85,B 0,C 180,E1 -12326.773,E2 -12326.773} C_VEL
LIN {X 0,Y 374.517,Z 783.881,A -85,B 0,C 180,E1 -12328.925,E2 -12328.925} C_VEL
LIN {X 0,Y 374.554,Z 784.137,A -85,B 0,C 180,E1 -12330,E2 -12330} C_VEL
LIN {X 0,Y 374.516,Z 783.983,A -85,B 0,C 180,E1 -12331.076,E2 -12331.076} C_VEL
LIN {X 0,Y 374.46,Z 782.412,A -85,B 0,C 180,E1 -12333.228,E2 -12333.228} C_VEL
LIN {X 0,Y 374.56,Z 781.032,A -85,B 0,C 180,E1 -12334.305,E2 -12334.305} C_VEL
LIN {X 0,Y 374.627,Z 777.694,A -85,B 0,C 180,E1 -12336.13,E2 -12336.13} C_VEL
LIN {X 0,Y 374.942,Z 772.606,A -85,B 0,C 180,E1 -12338.082,E2 -12338.082} C_VEL
LIN {X 0,Y 375.485,Z 766.085,A -85,B 0,C 180,E1 -12339.97,E2 -12339.97} C_VEL
LIN {X 0,Y 376.117,Z 758.981,A -85,B 0,C 180,E1 -12341.588,E2 -12341.588} C_VEL
LIN {X 0,Y 377.111,Z 750.135,A -85,B 0,C 180,E1 -12343.197,E2 -12343.197} C_VEL
LIN {X 0,Y 377.995,Z 740.463,A -85,B 0,C 180,E1 -12344.628,E2 -12344.628} C_VEL
LIN {X 0,Y 378.998,Z 729.961,A -85,B 0,C 180,E1 -12345.874,E2 -12345.874} C_VEL
LIN {X 0,Y 380.095,Z 718.766,A -85,B 0,C 180,E1 -12346.931,E2 -12346.931} C_VEL
LIN {X 0,Y 380.649,Z 711.068,A -85,B 0,C 180,E1 -12347.536,E2 -12347.536} C_VEL
LIN {X 0,Y 379.392,Z 698.425,A -85,B 0,C 180,E1 -12348.426,E2 -12348.426} C_VEL
LIN {X 0,Y 377.135,Z 685.525,A -85,B 0,C 180,E1 -12349.167,E2 -12349.167} C_VEL
LIN {X 0,Y 375.264,Z 676.936,A -85,B 0,C 180,E1 -12349.58,E2 -12349.58} C_VEL
LIN {X 0,Y 375.597,Z 671.341,A -85,B 0,C 180,E1 -12352.556,E2 -12352.556} C_VEL
LIN {X 0,Y 375.987,Z 664.687,A -85,B 0,C 180,E1 -12356.204,E2 -12356.204} C_VEL
LIN {X 0,Y 376.51,Z 658.658,A -85,B 0,C 180,E1 -12359.647,E2 -12359.647} C_VEL
LIN {X 0,Y 377.09,Z 653.041,A -85,B 0,C 180,E1 -12362.998,E2 -12362.998} C_VEL
LIN {X 0,Y 377.443,Z 648.439,A -85,B 0,C 180,E1 -12365.911,E2 -12365.911} C_VEL
LIN {X 0,Y 377.129,Z 644.694,A -85,B 0,C 180,E1 -12368.492,E2 -12368.492} C_VEL
LIN {X 0,Y 376.412,Z 640.459,A -85,B 0,C 180,E1 -12371.682,E2 -12371.682} C_VEL
LIN {X 0,Y 375.993,Z 637.652,A -85,B 0,C 180,E1 -12373.994,E2 -12373.994} C_VEL
LIN {X 0,Y 375.933,Z 637.66,A -85,B 0,C 180,E1 -12377.7,E2 -12377.7} C_VEL
LIN {X 0,Y 375.964,Z 637.657,A -85,B 0,C 180,E1 -12380.538,E2 -12380.538} C_VEL
LIN {X 0,Y 375.965,Z 637.656,A -85,B 0,C 180,E1 -12383.496,E2 -12383.496} C_VEL
LIN {X 0,Y 375.961,Z 637.654,A -85,B 0,C 180,E1 -12385.889,E2 -12385.889} C_VEL
LIN {X 0,Y 375.966,Z 637.653,A -85,B 0,C 180,E1 -12389.687,E2 -12389.687} C_VEL
LIN {X 0,Y 376.021,Z 637.646,A -85,B 0,C 180,E1 -12393.348,E2 -12393.348} C_VEL
LIN {X 0,Y 375.998,Z 637.651,A -85,B 0,C 180,E1 -12396.888,E2 -12396.888} C_VEL
LIN {X 0,Y 376,Z 637.65,A -85,B 0,C 180,E1 -12400.339,E2 -12400.339} C_VEL
LIN {X 0,Y 376.031,Z 637.647,A -85,B 0,C 180,E1 -12403.719,E2 -12403.719} C_VEL
LIN {X 0,Y 376.105,Z 637.637,A -85,B 0,C 180,E1 -12407.042,E2 -12407.042} C_VEL
LIN {X 0,Y 376.121,Z 637.633,A -85,B 0,C 180,E1 -12410.319,E2 -12410.319} C_VEL
LIN {X 0,Y 376.232,Z 637.62,A -85,B 0,C 180,E1 -12412.487,E2 -12412.487} C_VEL
LIN {X 0,Y 376.173,Z 637.629,A -85,B 0,C 180,E1 -12414.64,E2 -12414.64} C_VEL
LIN {X 0,Y 376.354,Z 637.607,A -85,B 0,C 180,E1 -12417.86,E2 -12417.86} C_VEL
LIN {X 0,Y 376.491,Z 637.59,A -85,B 0,C 180,E1 -12420,E2 -12420} C_VEL
LIN {X 0,Y 376.192,Z 637.629,A -85,B 0,C 180,E1 -12423.213,E2 -12423.213} C_VEL
LIN {X 0,Y 376.246,Z 637.73,A -85,B 0,C 180,E1 -12426.624,E2 -12426.624} C_VEL
LIN {X 0,Y 376.343,Z 638.915,A -85,B 0,C 180,E1 -12428.211,E2 -12428.211} C_VEL
LIN {X 0,Y 376.213,Z 641.52,A -85,B 0,C 180,E1 -12430.767,E2 -12430.767} C_VEL
LIN {X 0,Y 375.919,Z 645.072,A -85,B 0,C 180,E1 -12434.066,E2 -12434.066} C_VEL
LIN {X 0,Y 375.654,Z 648.801,A -85,B 0,C 180,E1 -12437.418,E2 -12437.418} C_VEL
LIN {X 0,Y 375.364,Z 652.754,A -85,B 0,C 180,E1 -12440.839,E2 -12440.839} C_VEL
LIN {X 0,Y 375.136,Z 656.937,A -85,B 0,C 180,E1 -12444.341,E2 -12444.341} C_VEL
LIN {X 0,Y 375.089,Z 658.335,A -85,B 0,C 180,E1 -12445.491,E2 -12445.491} C_VEL
LIN {X 0,Y 378.918,Z 672.736,A -85,B 0,C 180,E1 -12446.319,E2 -12446.319} C_VEL
LIN {X 0,Y 381.15,Z 684.316,A -85,B 0,C 180,E1 -12447.115,E2 -12447.115} C_VEL
LIN {X 0,Y 381.341,Z 688.718,A -85,B 0,C 180,E1 -12447.435,E2 -12447.435} C_VEL
LIN {X 0,Y 380.346,Z 700.689,A -85,B 0,C 180,E1 -12448.382,E2 -12448.382} C_VEL
LIN {X 0,Y 379.305,Z 712.379,A -85,B 0,C 180,E1 -12449.586,E2 -12449.586} C_VEL
LIN {X 0,Y 378.34,Z 721.323,A -85,B 0,C 180,E1 -12450.72,E2 -12450.72} C_VEL
LIN {X 0,Y 377.473,Z 729.926,A -85,B 0,C 180,E1 -12452.048,E2 -12452.048} C_VEL
LIN {X 0,Y 376.678,Z 737.5,A -85,B 0,C 180,E1 -12453.47,E2 -12453.47} C_VEL
LIN {X 0,Y 375.964,Z 744.228,A -85,B 0,C 180,E1 -12455.017,E2 -12455.017} C_VEL
LIN {X 0,Y 375.347,Z 750.373,A -85,B 0,C 180,E1 -12456.811,E2 -12456.811} C_VEL
LIN {X 0,Y 375.017,Z 754.163,A -85,B 0,C 180,E1 -12458.202,E2 -12458.202} C_VEL
LIN {X 0,Y 374.76,Z 757.419,A -85,B 0,C 180,E1 -12459.746,E2 -12459.746} C_VEL
LIN {X 0,Y 374.505,Z 759.836,A -85,B 0,C 180,E1 -12461.354,E2 -12461.354} C_VEL
LIN {X 0,Y 374.409,Z 761.303,A -85,B 0,C 180,E1 -12462.94,E2 -12462.94} C_VEL
LIN {X 0,Y 374.322,Z 761.899,A -85,B 0,C 180,E1 -12464.483,E2 -12464.483} C_VEL
LIN {X 0,Y 374.314,Z 761.698,A -85,B 0,C 180,E1 -12465.996,E2 -12465.996} C_VEL
LIN {X 0,Y 374.372,Z 760.742,A -85,B 0,C 180,E1 -12467.482,E2 -12467.482} C_VEL
LIN {X 0,Y 374.546,Z 758.997,A -85,B 0,C 180,E1 -12468.948,E2 -12468.948} C_VEL
LIN {X 0,Y 374.753,Z 756.536,A -85,B 0,C 180,E1 -12470.385,E2 -12470.385} C_VEL
LIN {X 0,Y 374.962,Z 753.012,A -85,B 0,C 180,E1 -12471.926,E2 -12471.926} C_VEL
LIN {X 0,Y 375.361,Z 747.952,A -85,B 0,C 180,E1 -12473.62,E2 -12473.62} C_VEL
LIN {X 0,Y 375.929,Z 741.376,A -85,B 0,C 180,E1 -12475.344,E2 -12475.344} C_VEL
LIN {X 0,Y 376.619,Z 734.176,A -85,B 0,C 180,E1 -12476.857,E2 -12476.857} C_VEL
LIN {X 0,Y 377.485,Z 724.883,A -85,B 0,C 180,E1 -12478.424,E2 -12478.424} C_VEL
LIN {X 0,Y 378.38,Z 715.181,A -85,B 0,C 180,E1 -12479.747,E2 -12479.747} C_VEL
LIN {X 0,Y 379.317,Z 704.524,A -85,B 0,C 180,E1 -12480.921,E2 -12480.921} C_VEL
LIN {X 0,Y 380.207,Z 692.508,A -85,B 0,C 180,E1 -12481.96,E2 -12481.96} C_VEL
LIN {X 0,Y 380.65,Z 684.726,A -85,B 0,C 180,E1 -12482.511,E2 -12482.511} C_VEL
LIN {X 0,Y 378.143,Z 671.737,A -85,B 0,C 180,E1 -12483.36,E2 -12483.36} C_VEL
LIN {X 0,Y 375.041,Z 658.265,A -85,B 0,C 180,E1 -12484.033,E2 -12484.033} C_VEL
LIN {X 0,Y 374.94,Z 657.463,A -85,B 0,C 180,E1 -12484.074,E2 -12484.074} C_VEL
LIN {X 0,Y 375.074,Z 652.45,A -85,B 0,C 180,E1 -12487.991,E2 -12487.991} C_VEL
LIN {X 0,Y 375.265,Z 649.559,A -85,B 0,C 180,E1 -12490.299,E2 -12490.299} C_VEL
LIN {X 0,Y 375.47,Z 645.374,A -85,B 0,C 180,E1 -12493.694,E2 -12493.694} C_VEL
LIN {X 0,Y 375.786,Z 641.34,A -85,B 0,C 180,E1 -12497.031,E2 -12497.031} C_VEL
LIN {X 0,Y 375.913,Z 637.661,A -85,B 0,C 180,E1 -12500.313,E2 -12500.313} C_VEL
LIN {X 0,Y 376.192,Z 637.624,A -85,B 0,C 180,E1 -12502.485,E2 -12502.485} C_VEL
LIN {X 0,Y 376.173,Z 637.628,A -85,B 0,C 180,E1 -12504.64,E2 -12504.64} C_VEL
LIN {X 0,Y 376.357,Z 637.601,A -85,B 0,C 180,E1 -12507.859,E2 -12507.859} C_VEL
LIN {X 0,Y 376.492,Z 637.585,A -85,B 0,C 180,E1 -12510,E2 -12510} C_VEL
LIN {X 0,Y 376.191,Z 637.625,A -85,B 0,C 180,E1 -12513.212,E2 -12513.212} C_VEL
LIN {X 0,Y 376.22,Z 637.621,A -85,B 0,C 180,E1 -12516.435,E2 -12516.435} C_VEL
LIN {X 0,Y 376.039,Z 637.645,A -85,B 0,C 180,E1 -12518.598,E2 -12518.598} C_VEL
LIN {X 0,Y 375.47,Z 637.8,A -85,B 0,C 180,E1 -12522.224,E2 -12522.224} C_VEL
LIN {X 0,Y 375.18,Z 643.825,A -85,B 0,C 180,E1 -12526.318,E2 -12526.318} C_VEL
LIN {X 0,Y 374.993,Z 648.831,A -85,B 0,C 180,E1 -12529.715,E2 -12529.715} C_VEL
LIN {X 0,Y 374.837,Z 654.073,A -85,B 0,C 180,E1 -12533.259,E2 -12533.259} C_VEL
LIN {X 0,Y 374.795,Z 654.862,A -85,B 0,C 180,E1 -12533.793,E2 -12533.793} C_VEL
LIN {X 0,Y 374.62,Z 656.459,A -85,B 0,C 180,E1 -12534.307,E2 -12534.307} C_VEL
LIN {X 0,Y 374.253,Z 659.094,A -85,B 0,C 180,E1 -12534.72,E2 -12534.72} C_VEL
LIN {X 0,Y 373.558,Z 664.153,A -85,B 0,C 180,E1 -12535.175,E2 -12535.175} C_VEL
LIN {X 0,Y 372.651,Z 674.855,A -85,B 0,C 180,E1 -12535.679,E2 -12535.679} C_VEL
LIN {X 0,Y 372.854,Z 680.524,A -85,B 0,C 180,E1 -12536.004,E2 -12536.004} C_VEL
LIN {X 0,Y 373.122,Z 682.338,A -85,B 0,C 180,E1 -12536.135,E2 -12536.135} C_VEL
LIN {X 0,Y 373.768,Z 686.6,A -85,B 0,C 180,E1 -12536.448,E2 -12536.448} C_VEL
LIN {X 0,Y 372.837,Z 698.684,A -85,B 0,C 180,E1 -12537.387,E2 -12537.387} C_VEL
LIN {X 0,Y 371.879,Z 709.894,A -85,B 0,C 180,E1 -12538.501,E2 -12538.501} C_VEL
LIN {X 0,Y 370.9,Z 720.491,A -85,B 0,C 180,E1 -12539.827,E2 -12539.827} C_VEL
LIN {X 0,Y 369.985,Z 729.737,A -85,B 0,C 180,E1 -12541.263,E2 -12541.263} C_VEL
LIN {X 0,Y 369.203,Z 738.1,A -85,B 0,C 180,E1 -12542.865,E2 -12542.865} C_VEL
LIN {X 0,Y 368.545,Z 745.078,A -85,B 0,C 180,E1 -12544.544,E2 -12544.544} C_VEL
LIN {X 0,Y 368.033,Z 750.845,A -85,B 0,C 180,E1 -12546.297,E2 -12546.297} C_VEL
LIN {X 0,Y 367.635,Z 756.003,A -85,B 0,C 180,E1 -12548.391,E2 -12548.391} C_VEL
LIN {X 0,Y 367.343,Z 758.904,A -85,B 0,C 180,E1 -12550.068,E2 -12550.068} C_VEL
LIN {X 0,Y 367.201,Z 761.038,A -85,B 0,C 180,E1 -12552.057,E2 -12552.057} C_VEL
LIN {X 0,Y 367.172,Z 761.78,A -85,B 0,C 180,E1 -12553.556,E2 -12553.556} C_VEL
LIN {X 0,Y 367.211,Z 761.772,A -85,B 0,C 180,E1 -12555.083,E2 -12555.083} C_VEL
LIN {X 0,Y 367.304,Z 760.931,A -85,B 0,C 180,E1 -12556.642,E2 -12556.642} C_VEL
LIN {X 0,Y 367.423,Z 759.225,A -85,B 0,C 180,E1 -12558.243,E2 -12558.243} C_VEL
LIN {X 0,Y 367.687,Z 756.58,A -85,B 0,C 180,E1 -12559.867,E2 -12559.867} C_VEL
LIN {X 0,Y 368.047,Z 752.86,A -85,B 0,C 180,E1 -12561.527,E2 -12561.527} C_VEL
LIN {X 0,Y 368.522,Z 747.892,A -85,B 0,C 180,E1 -12563.222,E2 -12563.222} C_VEL
LIN {X 0,Y 369.24,Z 741.517,A -85,B 0,C 180,E1 -12564.928,E2 -12564.928} C_VEL
LIN {X 0,Y 370.105,Z 733.278,A -85,B 0,C 180,E1 -12566.669,E2 -12566.669} C_VEL
LIN {X 0,Y 371.205,Z 724.019,A -85,B 0,C 180,E1 -12568.233,E2 -12568.233} C_VEL
LIN {X 0,Y 372.266,Z 713.977,A -85,B 0,C 180,E1 -12569.587,E2 -12569.587} C_VEL
LIN {X 0,Y 373.204,Z 703.97,A -85,B 0,C 180,E1 -12570.684,E2 -12570.684} C_VEL
LIN {X 0,Y 374.257,Z 692.609,A -85,B 0,C 180,E1 -12571.678,E2 -12571.678} C_VEL
LIN {X 0,Y 374.611,Z 687.81,A -85,B 0,C 180,E1 -12572.029,E2 -12572.029} C_VEL
LIN {X 0,Y 372.965,Z 677.374,A -85,B 0,C 180,E1 -12572.809,E2 -12572.809} C_VEL
LIN {X 0,Y 369.959,Z 664.779,A -85,B 0,C 180,E1 -12573.599,E2 -12573.599} C_VEL
LIN {X 0,Y 367.948,Z 657.484,A -85,B 0,C 180,E1 -12573.994,E2 -12573.994} C_VEL
LIN {X 0,Y 368.017,Z 652.268,A -85,B 0,C 180,E1 -12577.546,E2 -12577.546} C_VEL
LIN {X 0,Y 368.21,Z 647.017,A -85,B 0,C 180,E1 -12581.066,E2 -12581.066} C_VEL
LIN {X 0,Y 368.397,Z 641.917,A -85,B 0,C 180,E1 -12584.509,E2 -12584.509} C_VEL
LIN {X 0,Y 368.625,Z 638.577,A -85,B 0,C 180,E1 -12586.774,E2 -12586.774} C_VEL
LIN {X 0,Y 368.985,Z 638.524,A -85,B 0,C 180,E1 -12590.129,E2 -12590.129} C_VEL
LIN {X 0,Y 369.158,Z 638.506,A -85,B 0,C 180,E1 -12592.342,E2 -12592.342} C_VEL
LIN {X 0,Y 369.141,Z 638.507,A -85,B 0,C 180,E1 -12594.537,E2 -12594.537} C_VEL
LIN {X 0,Y 369.316,Z 638.483,A -85,B 0,C 180,E1 -12597.819,E2 -12597.819} C_VEL
LIN {X 0,Y 369.457,Z 638.466,A -85,B 0,C 180,E1 -12600,E2 -12600} C_VEL
LIN {X 0,Y 369.316,Z 638.483,A -85,B 0,C 180,E1 -12602.181,E2 -12602.181} C_VEL
LIN {X 0,Y 369.205,Z 638.498,A -85,B 0,C 180,E1 -12606.558,E2 -12606.558} C_VEL
LIN {X 0,Y 369.134,Z 638.506,A -85,B 0,C 180,E1 -12608.761,E2 -12608.761} C_VEL
LIN {X 0,Y 369.002,Z 638.52,A -85,B 0,C 180,E1 -12612.093,E2 -12612.093} C_VEL
LIN {X 0,Y 368.994,Z 638.524,A -85,B 0,C 180,E1 -12615.465,E2 -12615.465} C_VEL
LIN {X 0,Y 368.979,Z 638.523,A -85,B 0,C 180,E1 -12618.893,E2 -12618.893} C_VEL
LIN {X 0,Y 368.929,Z 638.531,A -85,B 0,C 180,E1 -12622.395,E2 -12622.395} C_VEL
LIN {X 0,Y 368.996,Z 638.521,A -85,B 0,C 180,E1 -12625.98,E2 -12625.98} C_VEL
LIN {X 0,Y 368.964,Z 638.524,A -85,B 0,C 180,E1 -12628.814,E2 -12628.814} C_VEL
LIN {X 0,Y 368.896,Z 638.536,A -85,B 0,C 180,E1 -12632.238,E2 -12632.238} C_VEL
LIN {X 0,Y 368.926,Z 638.532,A -85,B 0,C 180,E1 -12635.002,E2 -12635.002} C_VEL
LIN {X 0,Y 368.908,Z 638.534,A -85,B 0,C 180,E1 -12638.641,E2 -12638.641} C_VEL
LIN {X 0,Y 368.878,Z 638.535,A -85,B 0,C 180,E1 -12642.01,E2 -12642.01} C_VEL
LIN {X 0,Y 368.877,Z 638.538,A -85,B 0,C 180,E1 -12645.176,E2 -12645.176} C_VEL
LIN {X 0,Y 368.927,Z 638.537,A -85,B 0,C 180,E1 -12647.733,E2 -12647.733} C_VEL
LIN {X 0,Y 369.836,Z 643.671,A -85,B 0,C 180,E1 -12651.181,E2 -12651.181} C_VEL
LIN {X 0,Y 370.272,Z 648.046,A -85,B 0,C 180,E1 -12653.957,E2 -12653.957} C_VEL
LIN {X 0,Y 370.034,Z 652.586,A -85,B 0,C 180,E1 -12656.688,E2 -12656.688} C_VEL
LIN {X 0,Y 369.457,Z 658.94,A -85,B 0,C 180,E1 -12660.358,E2 -12660.358} C_VEL
LIN {X 0,Y 368.892,Z 665.467,A -85,B 0,C 180,E1 -12664.012,E2 -12664.012} C_VEL
LIN {X 0,Y 368.415,Z 673.047,A -85,B 0,C 180,E1 -12668.162,E2 -12668.162} C_VEL
LIN {X 0,Y 368.173,Z 677.11,A -85,B 0,C 180,E1 -12670.341,E2 -12670.341} C_VEL
LIN {X 0,Y 370.847,Z 690.916,A -85,B 0,C 180,E1 -12671.045,E2 -12671.045} C_VEL
LIN {X 0,Y 372.578,Z 703.555,A -85,B 0,C 180,E1 -12671.861,E2 -12671.861} C_VEL
LIN {X 0,Y 373.354,Z 711.481,A -85,B 0,C 180,E1 -12672.472,E2 -12672.472} C_VEL
LIN {X 0,Y 372.377,Z 722.676,A -85,B 0,C 180,E1 -12673.414,E2 -12673.414} C_VEL
LIN {X 0,Y 371.456,Z 732.833,A -85,B 0,C 180,E1 -12674.5,E2 -12674.5} C_VEL
LIN {X 0,Y 370.358,Z 744.384,A -85,B 0,C 180,E1 -12675.999,E2 -12675.999} C_VEL
LIN {X 0,Y 369.536,Z 752.896,A -85,B 0,C 180,E1 -12677.367,E2 -12677.367} C_VEL
LIN {X 0,Y 368.692,Z 761.197,A -85,B 0,C 180,E1 -12679.012,E2 -12679.012} C_VEL
LIN {X 0,Y 368.144,Z 767.89,A -85,B 0,C 180,E1 -12680.662,E2 -12680.662} C_VEL
LIN {X 0,Y 367.727,Z 773.221,A -85,B 0,C 180,E1 -12682.312,E2 -12682.312} C_VEL
LIN {X 0,Y 367.513,Z 777.305,A -85,B 0,C 180,E1 -12683.937,E2 -12683.937} C_VEL
LIN {X 0,Y 367.465,Z 780.434,A -85,B 0,C 180,E1 -12685.613,E2 -12685.613} C_VEL
LIN {X 0,Y 367.379,Z 781.946,A -85,B 0,C 180,E1 -12686.71,E2 -12686.71} C_VEL
LIN {X 0,Y 367.417,Z 783.657,A -85,B 0,C 180,E1 -12688.904,E2 -12688.904} C_VEL
LIN {X 0,Y 367.456,Z 783.921,A -85,B 0,C 180,E1 -12690,E2 -12690} C_VEL
LIN {X 0,Y 367.416,Z 783.78,A -85,B 0,C 180,E1 -12691.096,E2 -12691.096} C_VEL
LIN {X 0,Y 367.379,Z 782.224,A -85,B 0,C 180,E1 -12693.29,E2 -12693.29} C_VEL
LIN {X 0,Y 367.466,Z 780.851,A -85,B 0,C 180,E1 -12694.388,E2 -12694.388} C_VEL
LIN {X 0,Y 367.531,Z 777.855,A -85,B 0,C 180,E1 -12696.089,E2 -12696.089} C_VEL
LIN {X 0,Y 367.783,Z 774.034,A -85,B 0,C 180,E1 -12697.688,E2 -12697.688} C_VEL
LIN {X 0,Y 368.175,Z 768.981,A -85,B 0,C 180,E1 -12699.338,E2 -12699.338} C_VEL
LIN {X 0,Y 368.746,Z 762.65,A -85,B 0,C 180,E1 -12700.988,E2 -12700.988} C_VEL
LIN {X 0,Y 369.64,Z 754.751,A -85,B 0,C 180,E1 -12702.63,E2 -12702.63} C_VEL
LIN {X 0,Y 370.717,Z 744.936,A -85,B 0,C 180,E1 -12704.268,E2 -12704.268} C_VEL
LIN {X 0,Y 371.681,Z 734.788,A -85,B 0,C 180,E1 -12705.632,E2 -12705.632} C_VEL
LIN {X 0,Y 372.829,Z 723.382,A -85,B 0,C 180,E1 -12706.848,E2 -12706.848} C_VEL
LIN {X 0,Y 373.799,Z 712.832,A -85,B 0,C 180,E1 -12707.745,E2 -12707.745} C_VEL
LIN {X 0,Y 372.753,Z 700.154,A -85,B 0,C 180,E1 -12708.695,E2 -12708.695} C_VEL
LIN {X 0,Y 370.55,Z 687.161,A -85,B 0,C 180,E1 -12709.49,E2 -12709.49} C_VEL
LIN {X 0,Y 368.245,Z 676.679,A -85,B 0,C 180,E1 -12710.041,E2 -12710.041} C_VEL
LIN {X 0,Y 368.569,Z 671.227,A -85,B 0,C 180,E1 -12713.011,E2 -12713.011} C_VEL
LIN {X 0,Y 368.976,Z 665.096,A -85,B 0,C 180,E1 -12716.462,E2 -12716.462} C_VEL
LIN {X 0,Y 369.484,Z 659.653,A -85,B 0,C 180,E1 -12719.64,E2 -12719.64} C_VEL
LIN {X 0,Y 370.121,Z 653.475,A -85,B 0,C 180,E1 -12723.413,E2 -12723.413} C_VEL
LIN {X 0,Y 370.436,Z 649.458,A -85,B 0,C 180,E1 -12726.025,E2 -12726.025} C_VEL
LIN {X 0,Y 370.052,Z 645.465,A -85,B 0,C 180,E1 -12728.861,E2 -12728.861} C_VEL
LIN {X 0,Y 369.364,Z 641.34,A -85,B 0,C 180,E1 -12732.092,E2 -12732.092} C_VEL
LIN {X 0,Y 368.9,Z 638.536,A -85,B 0,C 180,E1 -12734.594,E2 -12734.594} C_VEL
LIN {X 0,Y 368.884,Z 638.539,A -85,B 0,C 180,E1 -12738.178,E2 -12738.178} C_VEL
LIN {X 0,Y 368.91,Z 638.535,A -85,B 0,C 180,E1 -12741.36,E2 -12741.36} C_VEL
LIN {X 0,Y 368.938,Z 638.531,A -85,B 0,C 180,E1 -12745.147,E2 -12745.147} C_VEL
LIN {X 0,Y 368.931,Z 638.531,A -85,B 0,C 180,E1 -12749.047,E2 -12749.047} C_VEL
LIN {X 0,Y 368.965,Z 638.527,A -85,B 0,C 180,E1 -12752.797,E2 -12752.797} C_VEL
LIN {X 0,Y 368.947,Z 638.525,A -85,B 0,C 180,E1 -12756.113,E2 -12756.113} C_VEL
LIN {X 0,Y 368.938,Z 638.53,A -85,B 0,C 180,E1 -12759.947,E2 -12759.947} C_VEL
LIN {X 0,Y 368.978,Z 638.526,A -85,B 0,C 180,E1 -12763.399,E2 -12763.399} C_VEL
LIN {X 0,Y 369.059,Z 638.516,A -85,B 0,C 180,E1 -12766.79,E2 -12766.79} C_VEL
LIN {X 0,Y 369.069,Z 638.511,A -85,B 0,C 180,E1 -12770.132,E2 -12770.132} C_VEL
LIN {X 0,Y 369.19,Z 638.496,A -85,B 0,C 180,E1 -12772.342,E2 -12772.342} C_VEL
LIN {X 0,Y 369.146,Z 638.503,A -85,B 0,C 180,E1 -12774.538,E2 -12774.538} C_VEL
LIN {X 0,Y 369.319,Z 638.483,A -85,B 0,C 180,E1 -12777.819,E2 -12777.819} C_VEL
LIN {X 0,Y 369.46,Z 638.466,A -85,B 0,C 180,E1 -12780,E2 -12780} C_VEL
LIN {X 0,Y 369.321,Z 638.485,A -85,B 0,C 180,E1 -12782.181,E2 -12782.181} C_VEL
LIN {X 0,Y 369.218,Z 638.598,A -85,B 0,C 180,E1 -12786.631,E2 -12786.631} C_VEL
LIN {X 0,Y 369.311,Z 640.612,A -85,B 0,C 180,E1 -12788.757,E2 -12788.757} C_VEL
LIN {X 0,Y 369.051,Z 643.994,A -85,B 0,C 180,E1 -12792.092,E2 -12792.092} C_VEL
LIN {X 0,Y 368.844,Z 646.375,A -85,B 0,C 180,E1 -12794.342,E2 -12794.342} C_VEL
LIN {X 0,Y 368.567,Z 650.138,A -85,B 0,C 180,E1 -12797.764,E2 -12797.764} C_VEL
LIN {X 0,Y 368.286,Z 654.124,A -85,B 0,C 180,E1 -12801.259,E2 -12801.259} C_VEL
LIN {X 0,Y 368.057,Z 658.635,A -85,B 0,C 180,E1 -12805.067,E2 -12805.067} C_VEL
LIN {X 0,Y 371.753,Z 672.023,A -85,B 0,C 180,E1 -12805.845,E2 -12805.845} C_VEL
LIN {X 0,Y 374.184,Z 684.1,A -85,B 0,C 180,E1 -12806.699,E2 -12806.699} C_VEL
LIN {X 0,Y 374.702,Z 688.657,A -85,B 0,C 180,E1 -12807.055,E2 -12807.055} C_VEL
LIN {X 0,Y 373.6,Z 701.071,A -85,B 0,C 180,E1 -12808.053,E2 -12808.053} C_VEL
LIN {X 0,Y 372.538,Z 712.225,A -85,B 0,C 180,E1 -12809.218,E2 -12809.218} C_VEL
LIN {X 0,Y 371.485,Z 721.786,A -85,B 0,C 180,E1 -12810.451,E2 -12810.451} C_VEL
LIN {X 0,Y 370.519,Z 730.962,A -85,B 0,C 180,E1 -12811.908,E2 -12811.908} C_VEL
LIN {X 0,Y 369.596,Z 738.882,A -85,B 0,C 180,E1 -12813.466,E2 -12813.466} C_VEL
LIN {X 0,Y 368.793,Z 746.101,A -85,B 0,C 180,E1 -12815.244,E2 -12815.244} C_VEL
LIN {X 0,Y 368.164,Z 752.148,A -85,B 0,C 180,E1 -12817.156,E2 -12817.156} C_VEL
LIN {X 0,Y 367.788,Z 756.646,A -85,B 0,C 180,E1 -12819.094,E2 -12819.094} C_VEL
LIN {X 0,Y 367.538,Z 759.14,A -85,B 0,C 180,E1 -12820.553,E2 -12820.553} C_VEL
LIN {X 0,Y 367.372,Z 760.867,A -85,B 0,C 180,E1 -12822.034,E2 -12822.034} C_VEL
LIN {X 0,Y 367.262,Z 761.869,A -85,B 0,C 180,E1 -12823.544,E2 -12823.544} C_VEL
LIN {X 0,Y 367.213,Z 762.129,A -85,B 0,C 180,E1 -12825.084,E2 -12825.084} C_VEL
LIN {X 0,Y 367.236,Z 761.591,A -85,B 0,C 180,E1 -12826.655,E2 -12826.655} C_VEL
LIN {X 0,Y 367.335,Z 760.163,A -85,B 0,C 180,E1 -12828.259,E2 -12828.259} C_VEL
LIN {X 0,Y 367.592,Z 757.804,A -85,B 0,C 180,E1 -12829.886,E2 -12829.886} C_VEL
LIN {X 0,Y 367.81,Z 754.344,A -85,B 0,C 180,E1 -12831.575,E2 -12831.575} C_VEL
LIN {X 0,Y 368.233,Z 749.682,A -85,B 0,C 180,E1 -12833.284,E2 -12833.284} C_VEL
LIN {X 0,Y 368.77,Z 743.142,A -85,B 0,C 180,E1 -12835.128,E2 -12835.128} C_VEL
LIN {X 0,Y 369.506,Z 735.565,A -85,B 0,C 180,E1 -12836.812,E2 -12836.812} C_VEL
LIN {X 0,Y 370.442,Z 726.087,A -85,B 0,C 180,E1 -12838.493,E2 -12838.493} C_VEL
LIN {X 0,Y 371.403,Z 716.402,A -85,B 0,C 180,E1 -12839.862,E2 -12839.862} C_VEL
LIN {X 0,Y 372.358,Z 705.814,A -85,B 0,C 180,E1 -12841.075,E2 -12841.075} C_VEL
LIN {X 0,Y 373.276,Z 694.451,A -85,B 0,C 180,E1 -12842.11,E2 -12842.11} C_VEL
LIN {X 0,Y 373.808,Z 686.112,A -85,B 0,C 180,E1 -12842.724,E2 -12842.724} C_VEL
LIN {X 0,Y 371.667,Z 674.524,A -85,B 0,C 180,E1 -12843.528,E2 -12843.528} C_VEL
LIN {X 0,Y 368.733,Z 661.555,A -85,B 0,C 180,E1 -12844.227,E2 -12844.227} C_VEL
LIN {X 0,Y 367.883,Z 657.62,A -85,B 0,C 180,E1 -12844.429,E2 -12844.429} C_VEL
LIN {X 0,Y 367.958,Z 653.706,A -85,B 0,C 180,E1 -12847.542,E2 -12847.542} C_VEL
LIN {X 0,Y 368.177,Z 650.781,A -85,B 0,C 180,E1 -12849.904,E2 -12849.904} C_VEL
LIN {X 0,Y 368.381,Z 646.552,A -85,B 0,C 180,E1 -12853.371,E2 -12853.371} C_VEL
LIN {X 0,Y 368.72,Z 642.504,A -85,B 0,C 180,E1 -12856.778,E2 -12856.778} C_VEL
LIN {X 0,Y 368.853,Z 638.632,A -85,B 0,C 180,E1 -12860.126,E2 -12860.126} C_VEL
LIN {X 0,Y 369.143,Z 638.501,A -85,B 0,C 180,E1 -12862.341,E2 -12862.341} C_VEL
LIN {X 0,Y 369.145,Z 638.502,A -85,B 0,C 180,E1 -12864.537,E2 -12864.537} C_VEL
LIN {X 0,Y 369.322,Z 638.477,A -85,B 0,C 180,E1 -12867.818,E2 -12867.818} C_VEL
LIN {X 0,Y 369.462,Z 638.46,A -85,B 0,C 180,E1 -12870,E2 -12870} C_VEL
LIN {X 0,Y 369.322,Z 638.478,A -85,B 0,C 180,E1 -12872.181,E2 -12872.181} C_VEL
LIN {X 0,Y 369.177,Z 638.499,A -85,B 0,C 180,E1 -12876.558,E2 -12876.558} C_VEL
LIN {X 0,Y 368.979,Z 638.526,A -85,B 0,C 180,E1 -12878.764,E2 -12878.764} C_VEL
LIN {X 0,Y 368.417,Z 638.658,A -85,B 0,C 180,E1 -12882.252,E2 -12882.252} C_VEL
LIN {X 0,Y 368.115,Z 645.078,A -85,B 0,C 180,E1 -12886.641,E2 -12886.641} C_VEL
LIN {X 0,Y 367.921,Z 650.138,A -85,B 0,C 180,E1 -12890.11,E2 -12890.11} C_VEL
LIN {X 0,Y 367.731,Z 656.188,A -85,B 0,C 180,E1 -12894.261,E2 -12894.261} C_VEL
LIN {X 0,Y 367.734,Z 656.861,A -85,B 0,C 180,E1 -12894.712,E2 -12894.712} C_VEL
LIN {X 0,Y 370.881,Z 670.687,A -85,B 0,C 180,E1 -12895.386,E2 -12895.386} C_VEL
LIN {X 0,Y 373.122,Z 682.338,A -85,B 0,C 180,E1 -12896.135,E2 -12896.135} C_VEL
LIN {X 0,Y 373.288,Z 686.021,A -85,B 0,C 180,E1 -12896.388,E2 -12896.388} C_VEL
LIN {X 0,Y 372.162,Z 691.413,A -85,B 0,C 180,E1 -12896.737,E2 -12896.737} C_VEL
LIN {X 0,Y 370.073,Z 696.574,A -85,B 0,C 180,E1 -12897.076,E2 -12897.076} C_VEL
LIN {X 0,Y 366.291,Z 704.897,A -85,B 0,C 180,E1 -12897.721,E2 -12897.721} C_VEL
LIN {X 0,Y 365.02,Z 709.761,A -85,B 0,C 180,E1 -12898.209,E2 -12898.209} C_VEL
LIN {X 0,Y 364.105,Z 719.364,A -85,B 0,C 180,E1 -12899.408,E2 -12899.408} C_VEL
LIN {X 0,Y 363.137,Z 728.766,A -85,B 0,C 180,E1 -12900.854,E2 -12900.854} C_VEL
LIN {X 0,Y 362.212,Z 737.771,A -85,B 0,C 180,E1 -12902.576,E2 -12902.576} C_VEL
LIN {X 0,Y 361.536,Z 744.971,A -85,B 0,C 180,E1 -12904.314,E2 -12904.314} C_VEL
LIN {X 0,Y 360.91,Z 751.536,A -85,B 0,C 180,E1 -12906.357,E2 -12906.357} C_VEL
LIN {X 0,Y 360.61,Z 755.255,A -85,B 0,C 180,E1 -12907.872,E2 -12907.872} C_VEL
LIN {X 0,Y 360.353,Z 758.093,A -85,B 0,C 180,E1 -12909.371,E2 -12909.371} C_VEL
LIN {X 0,Y 360.127,Z 760.866,A -85,B 0,C 180,E1 -12911.568,E2 -12911.568} C_VEL
LIN {X 0,Y 360.08,Z 762.008,A -85,B 0,C 180,E1 -12913.766,E2 -12913.766} C_VEL
LIN {X 0,Y 360.121,Z 761.887,A -85,B 0,C 180,E1 -12915.367,E2 -12915.367} C_VEL
LIN {X 0,Y 360.233,Z 760.98,A -85,B 0,C 180,E1 -12916.934,E2 -12916.934} C_VEL
LIN {X 0,Y 360.354,Z 759.299,A -85,B 0,C 180,E1 -12918.463,E2 -12918.463} C_VEL
LIN {X 0,Y 360.618,Z 756.861,A -85,B 0,C 180,E1 -12919.974,E2 -12919.974} C_VEL
LIN {X 0,Y 360.964,Z 753.675,A -85,B 0,C 180,E1 -12921.461,E2 -12921.461} C_VEL
LIN {X 0,Y 361.485,Z 748.571,A -85,B 0,C 180,E1 -12923.284,E2 -12923.284} C_VEL
LIN {X 0,Y 362.147,Z 742.737,A -85,B 0,C 180,E1 -12924.918,E2 -12924.918} C_VEL
LIN {X 0,Y 362.983,Z 735.299,A -85,B 0,C 180,E1 -12926.595,E2 -12926.595} C_VEL
LIN {X 0,Y 364.066,Z 726.703,A -85,B 0,C 180,E1 -12928.143,E2 -12928.143} C_VEL
LIN {X 0,Y 365.246,Z 716.272,A -85,B 0,C 180,E1 -12929.663,E2 -12929.663} C_VEL
LIN {X 0,Y 366.303,Z 705.897,A -85,B 0,C 180,E1 -12930.866,E2 -12930.866} C_VEL
LIN {X 0,Y 367.482,Z 693.693,A -85,B 0,C 180,E1 -12931.982,E2 -12931.982} C_VEL
LIN {X 0,Y 367.84,Z 688.253,A -85,B 0,C 180,E1 -12932.398,E2 -12932.398} C_VEL
LIN {X 0,Y 365.724,Z 676.085,A -85,B 0,C 180,E1 -12933.327,E2 -12933.327} C_VEL
LIN {X 0,Y 362.57,Z 663.688,A -85,B 0,C 180,E1 -12934.119,E2 -12934.119} C_VEL
LIN {X 0,Y 360.95,Z 657.662,A -85,B 0,C 180,E1 -12934.448,E2 -12934.448} C_VEL
LIN {X 0,Y 360.996,Z 652.079,A -85,B 0,C 180,E1 -12938.29,E2 -12938.29} C_VEL
LIN {X 0,Y 361.201,Z 646.836,A -85,B 0,C 180,E1 -12941.861,E2 -12941.861} C_VEL
LIN {X 0,Y 361.428,Z 641.633,A -85,B 0,C 180,E1 -12945.357,E2 -12945.357} C_VEL
LIN {X 0,Y 361.609,Z 639.451,A -85,B 0,C 180,E1 -12946.942,E2 -12946.942} C_VEL
LIN {X 0,Y 361.915,Z 639.405,A -85,B 0,C 180,E1 -12949.935,E2 -12949.935} C_VEL
LIN {X 0,Y 362.113,Z 639.383,A -85,B 0,C 180,E1 -12952.192,E2 -12952.192} C_VEL
LIN {X 0,Y 362.113,Z 639.382,A -85,B 0,C 180,E1 -12954.431,E2 -12954.431} C_VEL
LIN {X 0,Y 362.28,Z 639.359,A -85,B 0,C 180,E1 -12957.776,E2 -12957.776} C_VEL
LIN {X 0,Y 362.426,Z 639.342,A -85,B 0,C 180,E1 -12960,E2 -12960} C_VEL
LIN {X 0,Y 362.28,Z 639.359,A -85,B 0,C 180,E1 -12962.224,E2 -12962.224} C_VEL
LIN {X 0,Y 362.168,Z 639.374,A -85,B 0,C 180,E1 -12966.686,E2 -12966.686} C_VEL
LIN {X 0,Y 362.07,Z 639.386,A -85,B 0,C 180,E1 -12968.933,E2 -12968.933} C_VEL
LIN {X 0,Y 361.957,Z 639.398,A -85,B 0,C 180,E1 -12972.332,E2 -12972.332} C_VEL
LIN {X 0,Y 361.958,Z 639.398,A -85,B 0,C 180,E1 -12974.621,E2 -12974.621} C_VEL
LIN {X 0,Y 361.956,Z 639.4,A -85,B 0,C 180,E1 -12978.1,E2 -12978.1} C_VEL
LIN {X 0,Y 361.888,Z 639.405,A -85,B 0,C 180,E1 -12981.653,E2 -12981.653} C_VEL
LIN {X 0,Y 361.925,Z 639.403,A -85,B 0,C 180,E1 -12985.29,E2 -12985.29} C_VEL
LIN {X 0,Y 361.919,Z 639.405,A -85,B 0,C 180,E1 -12987.778,E2 -12987.778} C_VEL
LIN {X 0,Y 361.844,Z 639.413,A -85,B 0,C 180,E1 -12991.286,E2 -12991.286} C_VEL
LIN {X 0,Y 361.851,Z 639.414,A -85,B 0,C 180,E1 -12994.281,E2 -12994.281} C_VEL
LIN {X 0,Y 361.862,Z 639.411,A -85,B 0,C 180,E1 -12997.224,E2 -12997.224} C_VEL
LIN {X 0,Y 361.833,Z 639.416,A -85,B 0,C 180,E1 -13000.756,E2 -13000.756} C_VEL
LIN {X 0,Y 361.815,Z 639.418,A -85,B 0,C 180,E1 -13004.369,E2 -13004.369} C_VEL
LIN {X 0,Y 361.896,Z 639.51,A -85,B 0,C 180,E1 -13007.558,E2 -13007.558} C_VEL
LIN {X 0,Y 362.749,Z 644.233,A -85,B 0,C 180,E1 -13010.803,E2 -13010.803} C_VEL
LIN {X 0,Y 363.171,Z 647.804,A -85,B 0,C 180,E1 -13013.138,E2 -13013.138} C_VEL
LIN {X 0,Y 363.197,Z 651.08,A -85,B 0,C 180,E1 -13015.192,E2 -13015.192} C_VEL
LIN {X 0,Y 362.648,Z 656.631,A -85,B 0,C 180,E1 -13018.508,E2 -13018.508} C_VEL
LIN {X 0,Y 362.175,Z 661.95,A -85,B 0,C 180,E1 -13021.614,E2 -13021.614} C_VEL
LIN {X 0,Y 361.637,Z 668.463,A -85,B 0,C 180,E1 -13025.303,E2 -13025.303} C_VEL
LIN {X 0,Y 361.33,Z 673.875,A -85,B 0,C 180,E1 -13028.312,E2 -13028.312} C_VEL
LIN {X 0,Y 361.137,Z 676.995,A -85,B 0,C 180,E1 -13029.905,E2 -13029.905} C_VEL
LIN {X 0,Y 363.819,Z 689.823,A -85,B 0,C 180,E1 -13030.566,E2 -13030.566} C_VEL
LIN {X 0,Y 365.651,Z 702.959,A -85,B 0,C 180,E1 -13031.43,E2 -13031.43} C_VEL
LIN {X 0,Y 366.488,Z 713.54,A -85,B 0,C 180,E1 -13032.277,E2 -13032.277} C_VEL
LIN {X 0,Y 365.335,Z 725.612,A -85,B 0,C 180,E1 -13033.373,E2 -13033.373} C_VEL
LIN {X 0,Y 364.29,Z 736.008,A -85,B 0,C 180,E1 -13034.578,E2 -13034.578} C_VEL
LIN {X 0,Y 363.233,Z 745.933,A -85,B 0,C 180,E1 -13036.004,E2 -13036.004} C_VEL
LIN {X 0,Y 362.271,Z 755.475,A -85,B 0,C 180,E1 -13037.679,E2 -13037.679} C_VEL
LIN {X 0,Y 361.508,Z 763.254,A -85,B 0,C 180,E1 -13039.358,E2 -13039.358} C_VEL
LIN {X 0,Y 360.953,Z 769.478,A -85,B 0,C 180,E1 -13041.039,E2 -13041.039} C_VEL
LIN {X 0,Y 360.594,Z 774.417,A -85,B 0,C 180,E1 -13042.722,E2 -13042.722} C_VEL
LIN {X 0,Y 360.399,Z 778.215,A -85,B 0,C 180,E1 -13044.405,E2 -13044.405} C_VEL
LIN {X 0,Y 360.374,Z 780.17,A -85,B 0,C 180,E1 -13045.526,E2 -13045.526} C_VEL
LIN {X 0,Y 360.3,Z 781.697,A -85,B 0,C 180,E1 -13046.646,E2 -13046.646} C_VEL
LIN {X 0,Y 360.263,Z 782.764,A -85,B 0,C 180,E1 -13047.764,E2 -13047.764} C_VEL
LIN {X 0,Y 360.317,Z 783.43,A -85,B 0,C 180,E1 -13048.883,E2 -13048.883} C_VEL
LIN {X 0,Y 360.36,Z 783.704,A -85,B 0,C 180,E1 -13050,E2 -13050} C_VEL
LIN {X 0,Y 360.315,Z 783.577,A -85,B 0,C 180,E1 -13051.118,E2 -13051.118} C_VEL
LIN {X 0,Y 360.3,Z 782.046,A -85,B 0,C 180,E1 -13053.355,E2 -13053.355} C_VEL
LIN {X 0,Y 360.376,Z 780.683,A -85,B 0,C 180,E1 -13054.474,E2 -13054.474} C_VEL
LIN {X 0,Y 360.448,Z 777.984,A -85,B 0,C 180,E1 -13056.067,E2 -13056.067} C_VEL
LIN {X 0,Y 360.719,Z 773.906,A -85,B 0,C 180,E1 -13057.839,E2 -13057.839} C_VEL
LIN {X 0,Y 361.129,Z 768.873,A -85,B 0,C 180,E1 -13059.522,E2 -13059.522} C_VEL
LIN {X 0,Y 361.734,Z 762.566,A -85,B 0,C 180,E1 -13061.203,E2 -13061.203} C_VEL
LIN {X 0,Y 362.697,Z 754.708,A -85,B 0,C 180,E1 -13062.876,E2 -13062.876} C_VEL
LIN {X 0,Y 363.642,Z 746.714,A -85,B 0,C 180,E1 -13064.266,E2 -13064.266} C_VEL
LIN {X 0,Y 364.707,Z 735.963,A -85,B 0,C 180,E1 -13065.795,E2 -13065.795} C_VEL
LIN {X 0,Y 365.892,Z 724.977,A -85,B 0,C 180,E1 -13067.033,E2 -13067.033} C_VEL
LIN {X 0,Y 367.022,Z 713.186,A -85,B 0,C 180,E1 -13068.081,E2 -13068.081} C_VEL
LIN {X 0,Y 365.963,Z 700.723,A -85,B 0,C 180,E1 -13069.055,E2 -13069.055} C_VEL
LIN {X 0,Y 363.835,Z 688.24,A -85,B 0,C 180,E1 -13069.859,E2 -13069.859} C_VEL
LIN {X 0,Y 361.197,Z 676.444,A -85,B 0,C 180,E1 -13070.502,E2 -13070.502} C_VEL
LIN {X 0,Y 361.483,Z 672.188,A -85,B 0,C 180,E1 -13072.883,E2 -13072.883} C_VEL
LIN {X 0,Y 361.944,Z 665.851,A -85,B 0,C 180,E1 -13076.526,E2 -13076.526} C_VEL
LIN {X 0,Y 362.384,Z 661.323,A -85,B 0,C 180,E1 -13079.223,E2 -13079.223} C_VEL
LIN {X 0,Y 362.991,Z 655.509,A -85,B 0,C 180,E1 -13082.828,E2 -13082.828} C_VEL
LIN {X 0,Y 363.39,Z 651.487,A -85,B 0,C 180,E1 -13085.465,E2 -13085.465} C_VEL
LIN {X 0,Y 363.175,Z 647.556,A -85,B 0,C 180,E1 -13088.262,E2 -13088.262} C_VEL
LIN {X 0,Y 362.596,Z 643.769,A -85,B 0,C 180,E1 -13091.224,E2 -13091.224} C_VEL
LIN {X 0,Y 361.997,Z 640.136,A -85,B 0,C 180,E1 -13094.341,E2 -13094.341} C_VEL
LIN {X 0,Y 361.865,Z 639.412,A -85,B 0,C 180,E1 -13095.148,E2 -13095.148} C_VEL
LIN {X 0,Y 361.829,Z 639.418,A -85,B 0,C 180,E1 -13098.669,E2 -13098.669} C_VEL
LIN {X 0,Y 361.87,Z 639.411,A -85,B 0,C 180,E1 -13101.575,E2 -13101.575} C_VEL
LIN {X 0,Y 361.876,Z 639.409,A -85,B 0,C 180,E1 -13104.655,E2 -13104.655} C_VEL
LIN {X 0,Y 361.839,Z 639.414,A -85,B 0,C 180,E1 -13108.371,E2 -13108.371} C_VEL
LIN {X 0,Y 361.91,Z 639.405,A -85,B 0,C 180,E1 -13112.221,E2 -13112.221} C_VEL
LIN {X 0,Y 361.93,Z 639.404,A -85,B 0,C 180,E1 -13114.71,E2 -13114.71} C_VEL
LIN {X 0,Y 361.894,Z 639.408,A -85,B 0,C 180,E1 -13118.347,E2 -13118.347} C_VEL
LIN {X 0,Y 361.969,Z 639.399,A -85,B 0,C 180,E1 -13122.061,E2 -13122.061} C_VEL
LIN {X 0,Y 362,Z 639.394,A -85,B 0,C 180,E1 -13126.101,E2 -13126.101} C_VEL
LIN {X 0,Y 362.033,Z 639.387,A -85,B 0,C 180,E1 -13129.938,E2 -13129.938} C_VEL
LIN {X 0,Y 362.153,Z 639.373,A -85,B 0,C 180,E1 -13132.193,E2 -13132.193} C_VEL
LIN {X 0,Y 362.12,Z 639.378,A -85,B 0,C 180,E1 -13134.431,E2 -13134.431} C_VEL
LIN {X 0,Y 362.283,Z 639.359,A -85,B 0,C 180,E1 -13137.776,E2 -13137.776} C_VEL
LIN {X 0,Y 362.43,Z 639.341,A -85,B 0,C 180,E1 -13140,E2 -13140} C_VEL
LIN {X 0,Y 362.285,Z 639.361,A -85,B 0,C 180,E1 -13142.224,E2 -13142.224} C_VEL
LIN {X 0,Y 362.12,Z 639.38,A -85,B 0,C 180,E1 -13145.569,E2 -13145.569} C_VEL
LIN {X 0,Y 362.231,Z 639.853,A -85,B 0,C 180,E1 -13146.685,E2 -13146.685} C_VEL
LIN {X 0,Y 362.308,Z 641.933,A -85,B 0,C 180,E1 -13148.927,E2 -13148.927} C_VEL
LIN {X 0,Y 362.009,Z 645.322,A -85,B 0,C 180,E1 -13152.331,E2 -13152.331} C_VEL
LIN {X 0,Y 361.774,Z 647.719,A -85,B 0,C 180,E1 -13154.628,E2 -13154.628} C_VEL
LIN {X 0,Y 361.486,Z 651.479,A -85,B 0,C 180,E1 -13158.124,E2 -13158.124} C_VEL
LIN {X 0,Y 361.193,Z 655.5,A -85,B 0,C 180,E1 -13161.697,E2 -13161.697} C_VEL
LIN {X 0,Y 361.035,Z 658.846,A -85,B 0,C 180,E1 -13164.588,E2 -13164.588} C_VEL
LIN {X 0,Y 365.142,Z 673.698,A -85,B 0,C 180,E1 -13165.51,E2 -13165.51} C_VEL
LIN {X 0,Y 367.525,Z 685.665,A -85,B 0,C 180,E1 -13166.398,E2 -13166.398} C_VEL
LIN {X 0,Y 367.993,Z 689.882,A -85,B 0,C 180,E1 -13166.744,E2 -13166.744} C_VEL
LIN {X 0,Y 366.993,Z 700.451,A -85,B 0,C 180,E1 -13167.611,E2 -13167.611} C_VEL
LIN {X 0,Y 365.956,Z 710.918,A -85,B 0,C 180,E1 -13168.693,E2 -13168.693} C_VEL
LIN {X 0,Y 364.728,Z 721.546,A -85,B 0,C 180,E1 -13170.066,E2 -13170.066} C_VEL
LIN {X 0,Y 363.721,Z 730.203,A -85,B 0,C 180,E1 -13171.447,E2 -13171.447} C_VEL
LIN {X 0,Y 362.703,Z 738.976,A -85,B 0,C 180,E1 -13173.179,E2 -13173.179} C_VEL
LIN {X 0,Y 361.927,Z 745.451,A -85,B 0,C 180,E1 -13174.775,E2 -13174.775} C_VEL
LIN {X 0,Y 361.328,Z 750.661,A -85,B 0,C 180,E1 -13176.365,E2 -13176.365} C_VEL
LIN {X 0,Y 360.932,Z 754.534,A -85,B 0,C 180,E1 -13177.833,E2 -13177.833} C_VEL
LIN {X 0,Y 360.649,Z 757.687,A -85,B 0,C 180,E1 -13179.378,E2 -13179.378} C_VEL
LIN {X 0,Y 360.453,Z 759.45,A -85,B 0,C 180,E1 -13180.499,E2 -13180.499} C_VEL
LIN {X 0,Y 360.28,Z 761.292,A -85,B 0,C 180,E1 -13182.16,E2 -13182.16} C_VEL
LIN {X 0,Y 360.15,Z 762.208,A -85,B 0,C 180,E1 -13183.778,E2 -13183.778} C_VEL
LIN {X 0,Y 360.113,Z 762.291,A -85,B 0,C 180,E1 -13185.365,E2 -13185.365} C_VEL
LIN {X 0,Y 360.166,Z 761.602,A -85,B 0,C 180,E1 -13186.924,E2 -13186.924} C_VEL
LIN {X 0,Y 360.26,Z 760.187,A -85,B 0,C 180,E1 -13188.449,E2 -13188.449} C_VEL
LIN {X 0,Y 360.504,Z 757.987,A -85,B 0,C 180,E1 -13189.959,E2 -13189.959} C_VEL
LIN {X 0,Y 360.71,Z 755.079,A -85,B 0,C 180,E1 -13191.429,E2 -13191.429} C_VEL
LIN {X 0,Y 361.152,Z 750.2,A -85,B 0,C 180,E1 -13193.299,E2 -13193.299} C_VEL
LIN {X 0,Y 361.554,Z 745.454,A -85,B 0,C 180,E1 -13194.727,E2 -13194.727} C_VEL
LIN {X 0,Y 362.285,Z 738.052,A -85,B 0,C 180,E1 -13196.529,E2 -13196.529} C_VEL
LIN {X 0,Y 363.144,Z 729.855,A -85,B 0,C 180,E1 -13198.113,E2 -13198.113} C_VEL
LIN {X 0,Y 364.058,Z 720.694,A -85,B 0,C 180,E1 -13199.552,E2 -13199.552} C_VEL
LIN {X 0,Y 365.144,Z 709.898,A -85,B 0,C 180,E1 -13200.922,E2 -13200.922} C_VEL
LIN {X 0,Y 366.044,Z 698.896,A -85,B 0,C 180,E1 -13202.031,E2 -13202.031} C_VEL
LIN {X 0,Y 366.96,Z 687.693,A -85,B 0,C 180,E1 -13202.919,E2 -13202.919} C_VEL
LIN {X 0,Y 364.827,Z 675.632,A -85,B 0,C 180,E1 -13203.793,E2 -13203.793} C_VEL
LIN {X 0,Y 361.935,Z 662.768,A -85,B 0,C 180,E1 -13204.523,E2 -13204.523} C_VEL
LIN {X 0,Y 360.81,Z 657.797,A -85,B 0,C 180,E1 -13204.78,E2 -13204.78} C_VEL
LIN {X 0,Y 360.952,Z 653.487,A -85,B 0,C 180,E1 -13208.287,E2 -13208.287} C_VEL
LIN {X 0,Y 361.205,Z 649.151,A -85,B 0,C 180,E1 -13211.861,E2 -13211.861} C_VEL
LIN {X 0,Y 361.5,Z 645.007,A -85,B 0,C 180,E1 -13215.36,E2 -13215.36} C_VEL
LIN {X 0,Y 361.694,Z 642.337,A -85,B 0,C 180,E1 -13217.658,E2 -13217.658} C_VEL
LIN {X 0,Y 361.812,Z 639.758,A -85,B 0,C 180,E1 -13219.931,E2 -13219.931} C_VEL
LIN {X 0,Y 362.097,Z 639.378,A -85,B 0,C 180,E1 -13222.191,E2 -13222.191} C_VEL
LIN {X 0,Y 362.118,Z 639.377,A -85,B 0,C 180,E1 -13224.431,E2 -13224.431} C_VEL
LIN {X 0,Y 362.286,Z 639.354,A -85,B 0,C 180,E1 -13227.776,E2 -13227.776} C_VEL
LIN {X 0,Y 362.431,Z 639.336,A -85,B 0,C 180,E1 -13230,E2 -13230} C_VEL
LIN {X 0,Y 362.286,Z 639.355,A -85,B 0,C 180,E1 -13232.223,E2 -13232.223} C_VEL
LIN {X 0,Y 362.136,Z 639.377,A -85,B 0,C 180,E1 -13236.686,E2 -13236.686} C_VEL
LIN {X 0,Y 361.913,Z 639.406,A -85,B 0,C 180,E1 -13238.937,E2 -13238.937} C_VEL
LIN {X 0,Y 361.356,Z 639.551,A -85,B 0,C 180,E1 -13242.281,E2 -13242.281} C_VEL
LIN {X 0,Y 361.065,Z 644.626,A -85,B 0,C 180,E1 -13245.813,E2 -13245.813} C_VEL
LIN {X 0,Y 360.875,Z 649.74,A -85,B 0,C 180,E1 -13249.333,E2 -13249.333} C_VEL
LIN {X 0,Y 360.696,Z 654.934,A -85,B 0,C 180,E1 -13252.935,E2 -13252.935} C_VEL
LIN {X 0,Y 360.682,Z 656.986,A -85,B 0,C 180,E1 -13254.345,E2 -13254.345} C_VEL
LIN {X 0,Y 364.114,Z 672.02,A -85,B 0,C 180,E1 -13255.127,E2 -13255.127} C_VEL
LIN {X 0,Y 366.534,Z 685.013,A -85,B 0,C 180,E1 -13256.015,E2 -13256.015} C_VEL
LIN {X 0,Y 366.852,Z 687.719,A -85,B 0,C 180,E1 -13256.219,E2 -13256.219} C_VEL
LIN {X 0,Y 365.952,Z 699.152,A -85,B 0,C 180,E1 -13257.136,E2 -13257.136} C_VEL
LIN {X 0,Y 365.02,Z 709.761,A -85,B 0,C 180,E1 -13258.209,E2 -13258.209} C_VEL
LIN {X 0,Y 363.883,Z 714.505,A -85,B 0,C 180,E1 -13258.736,E2 -13258.736} C_VEL
LIN {X 0,Y 360.38,Z 721.899,A -85,B 0,C 180,E1 -13259.623,E2 -13259.623} C_VEL
LIN {X 0,Y 356.878,Z 728.757,A -85,B 0,C 180,E1 -13260.62,E2 -13260.62} C_VEL
LIN {X 0,Y 355.754,Z 732.659,A -85,B 0,C 180,E1 -13261.31,E2 -13261.31} C_VEL
LIN {X 0,Y 354.985,Z 740.489,A -85,B 0,C 180,E1 -13262.972,E2 -13262.972} C_VEL
LIN {X 0,Y 354.268,Z 747.302,A -85,B 0,C 180,E1 -13264.773,E2 -13264.773} C_VEL
LIN {X 0,Y 353.758,Z 752.624,A -85,B 0,C 180,E1 -13266.583,E2 -13266.583} C_VEL
LIN {X 0,Y 353.512,Z 756.002,A -85,B 0,C 180,E1 -13268.045,E2 -13268.045} C_VEL
LIN {X 0,Y 353.245,Z 758.639,A -85,B 0,C 180,E1 -13269.542,E2 -13269.542} C_VEL
LIN {X 0,Y 353.062,Z 760.571,A -85,B 0,C 180,E1 -13271.062,E2 -13271.062} C_VEL
LIN {X 0,Y 352.997,Z 761.796,A -85,B 0,C 180,E1 -13272.603,E2 -13272.603} C_VEL
LIN {X 0,Y 352.994,Z 762.272,A -85,B 0,C 180,E1 -13274.213,E2 -13274.213} C_VEL
LIN {X 0,Y 353.054,Z 761.926,A -85,B 0,C 180,E1 -13275.835,E2 -13275.835} C_VEL
LIN {X 0,Y 353.179,Z 760.808,A -85,B 0,C 180,E1 -13277.423,E2 -13277.423} C_VEL
LIN {X 0,Y 353.391,Z 758.792,A -85,B 0,C 180,E1 -13279.087,E2 -13279.087} C_VEL
LIN {X 0,Y 353.716,Z 755.769,A -85,B 0,C 180,E1 -13280.794,E2 -13280.794} C_VEL
LIN {X 0,Y 354.168,Z 751.607,A -85,B 0,C 180,E1 -13282.536,E2 -13282.536} C_VEL
LIN {X 0,Y 354.951,Z 744.973,A -85,B 0,C 180,E1 -13284.641,E2 -13284.641} C_VEL
LIN {X 0,Y 355.817,Z 737.659,A -85,B 0,C 180,E1 -13286.423,E2 -13286.423} C_VEL
LIN {X 0,Y 356.795,Z 730.262,A -85,B 0,C 180,E1 -13287.885,E2 -13287.885} C_VEL
LIN {X 0,Y 357.851,Z 721.602,A -85,B 0,C 180,E1 -13289.294,E2 -13289.294} C_VEL
LIN {X 0,Y 358.957,Z 712.3,A -85,B 0,C 180,E1 -13290.534,E2 -13290.534} C_VEL
LIN {X 0,Y 360.033,Z 702.226,A -85,B 0,C 180,E1 -13291.627,E2 -13291.627} C_VEL
LIN {X 0,Y 361.107,Z 690.598,A -85,B 0,C 180,E1 -13292.626,E2 -13292.626} C_VEL
LIN {X 0,Y 359.985,Z 682.221,A -85,B 0,C 180,E1 -13293.318,E2 -13293.318} C_VEL
LIN {X 0,Y 357.333,Z 669.923,A -85,B 0,C 180,E1 -13294.205,E2 -13294.205} C_VEL
LIN {X 0,Y 353.891,Z 657.825,A -85,B 0,C 180,E1 -13294.96,E2 -13294.96} C_VEL
LIN {X 0,Y 354.031,Z 651.921,A -85,B 0,C 180,E1 -13299.064,E2 -13299.064} C_VEL
LIN {X 0,Y 354.241,Z 646.673,A -85,B 0,C 180,E1 -13302.687,E2 -13302.687} C_VEL
LIN {X 0,Y 354.565,Z 640.343,A -85,B 0,C 180,E1 -13306.987,E2 -13306.987} C_VEL
LIN {X 0,Y 354.974,Z 640.272,A -85,B 0,C 180,E1 -13310.887,E2 -13310.887} C_VEL
LIN {X 0,Y 355.122,Z 640.254,A -85,B 0,C 180,E1 -13313.18,E2 -13313.18} C_VEL
LIN {X 0,Y 355.243,Z 640.236,A -85,B 0,C 180,E1 -13317.732,E2 -13317.732} C_VEL
LIN {X 0,Y 355.396,Z 640.218,A -85,B 0,C 180,E1 -13320,E2 -13320} C_VEL
LIN {X 0,Y 355.243,Z 640.236,A -85,B 0,C 180,E1 -13322.268,E2 -13322.268} C_VEL
LIN {X 0,Y 355.134,Z 640.25,A -85,B 0,C 180,E1 -13326.819,E2 -13326.819} C_VEL
LIN {X 0,Y 355.011,Z 640.265,A -85,B 0,C 180,E1 -13329.112,E2 -13329.112} C_VEL
LIN {X 0,Y 354.918,Z 640.276,A -85,B 0,C 180,E1 -13332.581,E2 -13332.581} C_VEL
LIN {X 0,Y 354.885,Z 640.279,A -85,B 0,C 180,E1 -13336.096,E2 -13336.096} C_VEL
LIN {X 0,Y 354.903,Z 640.278,A -85,B 0,C 180,E1 -13338.472,E2 -13338.472} C_VEL
LIN {X 0,Y 354.831,Z 640.287,A -85,B 0,C 180,E1 -13342.106,E2 -13342.106} C_VEL
LIN {X 0,Y 354.896,Z 640.278,A -85,B 0,C 180,E1 -13345.828,E2 -13345.828} C_VEL
LIN {X 0,Y 354.851,Z 640.285,A -85,B 0,C 180,E1 -13349.679,E2 -13349.679} C_VEL
LIN {X 0,Y 354.803,Z 640.29,A -85,B 0,C 180,E1 -13353.702,E2 -13353.702} C_VEL
LIN {X 0,Y 354.796,Z 640.292,A -85,B 0,C 180,E1 -13356.46,E2 -13356.46} C_VEL
LIN {X 0,Y 354.821,Z 640.287,A -85,B 0,C 180,E1 -13359.424,E2 -13359.424} C_VEL
LIN {X 0,Y 354.785,Z 640.293,A -85,B 0,C 180,E1 -13362.868,E2 -13362.868} C_VEL
LIN {X 0,Y 354.812,Z 640.29,A -85,B 0,C 180,E1 -13367.129,E2 -13367.129} C_VEL
LIN {X 0,Y 355.643,Z 644.788,A -85,B 0,C 180,E1 -13370.416,E2 -13370.416} C_VEL
LIN {X 0,Y 356.125,Z 648.639,A -85,B 0,C 180,E1 -13372.994,E2 -13372.994} C_VEL
LIN {X 0,Y 356.188,Z 651.915,A -85,B 0,C 180,E1 -13375.097,E2 -13375.097} C_VEL
LIN {X 0,Y 355.642,Z 656.972,A -85,B 0,C 180,E1 -13378.184,E2 -13378.184} C_VEL
LIN {X 0,Y 355.302,Z 660.838,A -85,B 0,C 180,E1 -13380.498,E2 -13380.498} C_VEL
LIN {X 0,Y 354.728,Z 667.125,A -85,B 0,C 180,E1 -13384.16,E2 -13384.16} C_VEL
LIN {X 0,Y 354.292,Z 673.608,A -85,B 0,C 180,E1 -13387.859,E2 -13387.859} C_VEL
LIN {X 0,Y 354.103,Z 676.35,A -85,B 0,C 180,E1 -13389.397,E2 -13389.397} C_VEL
LIN {X 0,Y 357.051,Z 690.106,A -85,B 0,C 180,E1 -13390.152,E2 -13390.152} C_VEL
LIN {X 0,Y 358.883,Z 703.652,A -85,B 0,C 180,E1 -13391.076,E2 -13391.076} C_VEL
LIN {X 0,Y 359.723,Z 713.92,A -85,B 0,C 180,E1 -13391.932,E2 -13391.932} C_VEL
LIN {X 0,Y 358.691,Z 724.495,A -85,B 0,C 180,E1 -13392.909,E2 -13392.909} C_VEL
LIN {X 0,Y 357.536,Z 735.389,A -85,B 0,C 180,E1 -13394.177,E2 -13394.177} C_VEL
LIN {X 0,Y 356.326,Z 745.997,A -85,B 0,C 180,E1 -13395.727,E2 -13395.727} C_VEL
LIN {X 0,Y 355.301,Z 755.259,A -85,B 0,C 180,E1 -13397.433,E2 -13397.433} C_VEL
LIN {X 0,Y 354.383,Z 764.017,A -85,B 0,C 180,E1 -13399.43,E2 -13399.43} C_VEL
LIN {X 0,Y 353.748,Z 770.943,A -85,B 0,C 180,E1 -13401.431,E2 -13401.431} C_VEL
LIN {X 0,Y 353.417,Z 775.519,A -85,B 0,C 180,E1 -13403.148,E2 -13403.148} C_VEL
LIN {X 0,Y 353.33,Z 777.925,A -85,B 0,C 180,E1 -13404.293,E2 -13404.293} C_VEL
LIN {X 0,Y 353.287,Z 779.893,A -85,B 0,C 180,E1 -13405.437,E2 -13405.437} C_VEL
LIN {X 0,Y 353.222,Z 781.437,A -85,B 0,C 180,E1 -13406.578,E2 -13406.578} C_VEL
LIN {X 0,Y 353.172,Z 782.524,A -85,B 0,C 180,E1 -13407.72,E2 -13407.72} C_VEL
LIN {X 0,Y 353.217,Z 783.201,A -85,B 0,C 180,E1 -13408.86,E2 -13408.86} C_VEL
LIN {X 0,Y 353.263,Z 783.485,A -85,B 0,C 180,E1 -13410,E2 -13410} C_VEL
LIN {X 0,Y 353.215,Z 783.373,A -85,B 0,C 180,E1 -13411.141,E2 -13411.141} C_VEL
LIN {X 0,Y 353.17,Z 782.824,A -85,B 0,C 180,E1 -13412.281,E2 -13412.281} C_VEL
LIN {X 0,Y 353.222,Z 781.869,A -85,B 0,C 180,E1 -13413.423,E2 -13413.423} C_VEL
LIN {X 0,Y 353.29,Z 780.515,A -85,B 0,C 180,E1 -13414.564,E2 -13414.564} C_VEL
LIN {X 0,Y 353.342,Z 778.182,A -85,B 0,C 180,E1 -13416.008,E2 -13416.008} C_VEL
LIN {X 0,Y 353.674,Z 773.777,A -85,B 0,C 180,E1 -13417.996,E2 -13417.996} C_VEL
LIN {X 0,Y 354.09,Z 768.765,A -85,B 0,C 180,E1 -13419.713,E2 -13419.713} C_VEL
LIN {X 0,Y 354.734,Z 762.495,A -85,B 0,C 180,E1 -13421.427,E2 -13421.427} C_VEL
LIN {X 0,Y 355.754,Z 754.703,A -85,B 0,C 180,E1 -13423.132,E2 -13423.132} C_VEL
LIN {X 0,Y 356.752,Z 746.771,A -85,B 0,C 180,E1 -13424.547,E2 -13424.547} C_VEL
LIN {X 0,Y 357.747,Z 737.144,A -85,B 0,C 180,E1 -13425.964,E2 -13425.964} C_VEL
LIN {X 0,Y 358.982,Z 726.524,A -85,B 0,C 180,E1 -13427.225,E2 -13427.225} C_VEL
LIN {X 0,Y 360.223,Z 714.969,A -85,B 0,C 180,E1 -13428.31,E2 -13428.31} C_VEL
LIN {X 0,Y 359.379,Z 702.909,A -85,B 0,C 180,E1 -13429.302,E2 -13429.302} C_VEL
LIN {X 0,Y 357.373,Z 690.302,A -85,B 0,C 180,E1 -13430.179,E2 -13430.179} C_VEL
LIN {X 0,Y 354.511,Z 678.036,A -85,B 0,C 180,E1 -13430.889,E2 -13430.889} C_VEL
LIN {X 0,Y 354.215,Z 676.219,A -85,B 0,C 180,E1 -13430.985,E2 -13430.985} C_VEL
LIN {X 0,Y 354.656,Z 669.98,A -85,B 0,C 180,E1 -13434.592,E2 -13434.592} C_VEL
LIN {X 0,Y 355.208,Z 663.711,A -85,B 0,C 180,E1 -13438.35,E2 -13438.35} C_VEL
LIN {X 0,Y 355.894,Z 657.546,A -85,B 0,C 180,E1 -13442.221,E2 -13442.221} C_VEL
LIN {X 0,Y 356.351,Z 653.515,A -85,B 0,C 180,E1 -13444.886,E2 -13444.886} C_VEL
LIN {X 0,Y 356.259,Z 649.577,A -85,B 0,C 180,E1 -13447.702,E2 -13447.702} C_VEL
LIN {X 0,Y 355.738,Z 645.778,A -85,B 0,C 180,E1 -13450.689,E2 -13450.689} C_VEL
LIN {X 0,Y 355.153,Z 642.131,A -85,B 0,C 180,E1 -13453.837,E2 -13453.837} C_VEL
LIN {X 0,Y 354.791,Z 640.293,A -85,B 0,C 180,E1 -13455.584,E2 -13455.584} C_VEL
LIN {X 0,Y 354.79,Z 640.294,A -85,B 0,C 180,E1 -13459.179,E2 -13459.179} C_VEL
LIN {X 0,Y 354.809,Z 640.292,A -85,B 0,C 180,E1 -13462.403,E2 -13462.403} C_VEL
LIN {X 0,Y 354.814,Z 640.29,A -85,B 0,C 180,E1 -13464.941,E2 -13464.941} C_VEL
LIN {X 0,Y 354.795,Z 640.292,A -85,B 0,C 180,E1 -13468.405,E2 -13468.405} C_VEL
LIN {X 0,Y 354.848,Z 640.283,A -85,B 0,C 180,E1 -13471.619,E2 -13471.619} C_VEL
LIN {X 0,Y 354.901,Z 640.277,A -85,B 0,C 180,E1 -13474.173,E2 -13474.173} C_VEL
LIN {X 0,Y 354.836,Z 640.287,A -85,B 0,C 180,E1 -13477.894,E2 -13477.894} C_VEL
LIN {X 0,Y 354.925,Z 640.276,A -85,B 0,C 180,E1 -13481.891,E2 -13481.891} C_VEL
LIN {X 0,Y 354.944,Z 640.273,A -85,B 0,C 180,E1 -13485.981,E2 -13485.981} C_VEL
LIN {X 0,Y 354.98,Z 640.266,A -85,B 0,C 180,E1 -13489.736,E2 -13489.736} C_VEL
LIN {X 0,Y 355.116,Z 640.249,A -85,B 0,C 180,E1 -13492.037,E2 -13492.037} C_VEL
LIN {X 0,Y 355.094,Z 640.253,A -85,B 0,C 180,E1 -13494.321,E2 -13494.321} C_VEL
LIN {X 0,Y 355.246,Z 640.235,A -85,B 0,C 180,E1 -13497.732,E2 -13497.732} C_VEL
LIN {X 0,Y 355.399,Z 640.217,A -85,B 0,C 180,E1 -13500,E2 -13500} C_VEL
LIN {X 0,Y 355.248,Z 640.238,A -85,B 0,C 180,E1 -13502.268,E2 -13502.268} C_VEL
LIN {X 0,Y 355.1,Z 640.255,A -85,B 0,C 180,E1 -13505.679,E2 -13505.679} C_VEL
LIN {X 0,Y 355.321,Z 642.701,A -85,B 0,C 180,E1 -13508.519,E2 -13508.519} C_VEL
LIN {X 0,Y 355.098,Z 645.49,A -85,B 0,C 180,E1 -13511.415,E2 -13511.415} C_VEL
LIN {X 0,Y 354.859,Z 648.058,A -85,B 0,C 180,E1 -13513.963,E2 -13513.963} C_VEL
LIN {X 0,Y 354.473,Z 652.182,A -85,B 0,C 180,E1 -13517.884,E2 -13517.884} C_VEL
LIN {X 0,Y 354.209,Z 655.779,A -85,B 0,C 180,E1 -13521.165,E2 -13521.165} C_VEL
LIN {X 0,Y 354.007,Z 659.09,A -85,B 0,C 180,E1 -13524.102,E2 -13524.102} C_VEL
LIN {X 0,Y 357.918,Z 672.721,A -85,B 0,C 180,E1 -13524.972,E2 -13524.972} C_VEL
LIN {X 0,Y 360.195,Z 683.178,A -85,B 0,C 180,E1 -13525.761,E2 -13525.761} C_VEL
LIN {X 0,Y 361.316,Z 690.636,A -85,B 0,C 180,E1 -13526.387,E2 -13526.387} C_VEL
LIN {X 0,Y 360.252,Z 701.298,A -85,B 0,C 180,E1 -13527.287,E2 -13527.287} C_VEL
LIN {X 0,Y 359.113,Z 712.217,A -85,B 0,C 180,E1 -13528.462,E2 -13528.462} C_VEL
LIN {X 0,Y 358.003,Z 721.263,A -85,B 0,C 180,E1 -13529.655,E2 -13529.655} C_VEL
LIN {X 0,Y 356.864,Z 730.398,A -85,B 0,C 180,E1 -13531.129,E2 -13531.129} C_VEL
LIN {X 0,Y 356.016,Z 737.57,A -85,B 0,C 180,E1 -13532.543,E2 -13532.543} C_VEL
LIN {X 0,Y 355.018,Z 745.2,A -85,B 0,C 180,E1 -13534.394,E2 -13534.394} C_VEL
LIN {X 0,Y 354.377,Z 750.542,A -85,B 0,C 180,E1 -13536.031,E2 -13536.031} C_VEL
LIN {X 0,Y 353.828,Z 755.513,A -85,B 0,C 180,E1 -13538.006,E2 -13538.006} C_VEL
LIN {X 0,Y 353.53,Z 758.37,A -85,B 0,C 180,E1 -13539.505,E2 -13539.505} C_VEL
LIN {X 0,Y 353.281,Z 760.495,A -85,B 0,C 180,E1 -13541.033,E2 -13541.033} C_VEL
LIN {X 0,Y 353.154,Z 761.863,A -85,B 0,C 180,E1 -13542.58,E2 -13542.58} C_VEL
LIN {X 0,Y 353.054,Z 762.526,A -85,B 0,C 180,E1 -13544.223,E2 -13544.223} C_VEL
LIN {X 0,Y 353.015,Z 762.387,A -85,B 0,C 180,E1 -13545.829,E2 -13545.829} C_VEL
LIN {X 0,Y 353.115,Z 761.447,A -85,B 0,C 180,E1 -13547.427,E2 -13547.427} C_VEL
LIN {X 0,Y 353.283,Z 759.578,A -85,B 0,C 180,E1 -13549.109,E2 -13549.109} C_VEL
LIN {X 0,Y 353.546,Z 756.715,A -85,B 0,C 180,E1 -13550.829,E2 -13550.829} C_VEL
LIN {X 0,Y 353.856,Z 752.679,A -85,B 0,C 180,E1 -13552.604,E2 -13552.604} C_VEL
LIN {X 0,Y 354.366,Z 747.33,A -85,B 0,C 180,E1 -13554.404,E2 -13554.404} C_VEL
LIN {X 0,Y 355.038,Z 740.313,A -85,B 0,C 180,E1 -13556.242,E2 -13556.242} C_VEL
LIN {X 0,Y 355.862,Z 733.042,A -85,B 0,C 180,E1 -13557.776,E2 -13557.776} C_VEL
LIN {X 0,Y 356.843,Z 723.588,A -85,B 0,C 180,E1 -13559.399,E2 -13559.399} C_VEL
LIN {X 0,Y 357.906,Z 713.721,A -85,B 0,C 180,E1 -13560.755,E2 -13560.755} C_VEL
LIN {X 0,Y 358.898,Z 702.78,A -85,B 0,C 180,E1 -13561.967,E2 -13561.967} C_VEL
LIN {X 0,Y 359.892,Z 691.028,A -85,B 0,C 180,E1 -13562.997,E2 -13562.997} C_VEL
LIN {X 0,Y 360.084,Z 688.659,A -85,B 0,C 180,E1 -13563.17,E2 -13563.17} C_VEL
LIN {X 0,Y 357.896,Z 676.385,A -85,B 0,C 180,E1 -13564.092,E2 -13564.092} C_VEL
LIN {X 0,Y 355.056,Z 663.53,A -85,B 0,C 180,E1 -13564.852,E2 -13564.852} C_VEL
LIN {X 0,Y 353.736,Z 658.003,A -85,B 0,C 180,E1 -13565.144,E2 -13565.144} C_VEL
LIN {X 0,Y 353.96,Z 653.249,A -85,B 0,C 180,E1 -13569.059,E2 -13569.059} C_VEL
LIN {X 0,Y 354.224,Z 648.944,A -85,B 0,C 180,E1 -13572.686,E2 -13572.686} C_VEL
LIN {X 0,Y 354.551,Z 644.823,A -85,B 0,C 180,E1 -13576.239,E2 -13576.239} C_VEL
LIN {X 0,Y 354.771,Z 640.57,A -85,B 0,C 180,E1 -13580.018,E2 -13580.018} C_VEL
LIN {X 0,Y 354.864,Z 640.284,A -85,B 0,C 180,E1 -13580.883,E2 -13580.883} C_VEL
LIN {X 0,Y 355.119,Z 640.25,A -85,B 0,C 180,E1 -13583.18,E2 -13583.18} C_VEL
LIN {X 0,Y 355.249,Z 640.23,A -85,B 0,C 180,E1 -13587.732,E2 -13587.732} C_VEL
LIN {X 0,Y 355.401,Z 640.211,A -85,B 0,C 180,E1 -13590,E2 -13590} C_VEL
LIN {X 0,Y 355.249,Z 640.231,A -85,B 0,C 180,E1 -13592.267,E2 -13592.267} C_VEL
LIN {X 0,Y 355.095,Z 640.256,A -85,B 0,C 180,E1 -13596.82,E2 -13596.82} C_VEL
LIN {X 0,Y 354.837,Z 640.285,A -85,B 0,C 180,E1 -13599.116,E2 -13599.116} C_VEL
LIN {X 0,Y 354.308,Z 640.441,A -85,B 0,C 180,E1 -13602.311,E2 -13602.311} C_VEL
LIN {X 0,Y 353.98,Z 645.904,A -85,B 0,C 180,E1 -13606.138,E2 -13606.138} C_VEL
LIN {X 0,Y 353.777,Z 651.05,A -85,B 0,C 180,E1 -13609.737,E2 -13609.737} C_VEL
LIN {X 0,Y 353.604,Z 657.023,A -85,B 0,C 180,E1 -13613.898,E2 -13613.898} C_VEL
LIN {X 0,Y 353.613,Z 657.268,A -85,B 0,C 180,E1 -13614.007,E2 -13614.007} C_VEL
LIN {X 0,Y 356.765,Z 670.926,A -85,B 0,C 180,E1 -13614.707,E2 -13614.707} C_VEL
LIN {X 0,Y 359.113,Z 682.682,A -85,B 0,C 180,E1 -13615.502,E2 -13615.502} C_VEL
LIN {X 0,Y 359.965,Z 688.649,A -85,B 0,C 180,E1 -13615.971,E2 -13615.971} C_VEL
LIN {X 0,Y 359.027,Z 700.055,A -85,B 0,C 180,E1 -13616.915,E2 -13616.915} C_VEL
LIN {X 0,Y 357.971,Z 711.426,A -85,B 0,C 180,E1 -13618.111,E2 -13618.111} C_VEL
LIN {X 0,Y 356.943,Z 721.768,A -85,B 0,C 180,E1 -13619.487,E2 -13619.487} C_VEL
LIN {X 0,Y 355.899,Z 731.583,A -85,B 0,C 180,E1 -13621.104,E2 -13621.104} C_VEL
LIN {X 0,Y 355.754,Z 732.659,A -85,B 0,C 180,E1 -13621.31,E2 -13621.31} C_VEL
LIN {X 0,Y 354.651,Z 736.402,A -85,B 0,C 180,E1 -13622.032,E2 -13622.032} C_VEL
LIN {X 0,Y 351.258,Z 742.052,A -85,B 0,C 180,E1 -13623.234,E2 -13623.234} C_VEL
LIN {X 0,Y 347.965,Z 747.082,A -85,B 0,C 180,E1 -13624.526,E2 -13624.526} C_VEL
LIN {X 0,Y 347.035,Z 749.782,A -85,B 0,C 180,E1 -13625.379,E2 -13625.379} C_VEL
LIN {X 0,Y 346.504,Z 755.164,A -85,B 0,C 180,E1 -13627.479,E2 -13627.479} C_VEL
LIN {X 0,Y 346.168,Z 758.867,A -85,B 0,C 180,E1 -13629.512,E2 -13629.512} C_VEL
LIN {X 0,Y 345.943,Z 760.985,A -85,B 0,C 180,E1 -13631.264,E2 -13631.264} C_VEL
LIN {X 0,Y 345.903,Z 762.383,A -85,B 0,C 180,E1 -13633.693,E2 -13633.693} C_VEL
LIN {X 0,Y 345.928,Z 762.356,A -85,B 0,C 180,E1 -13635.321,E2 -13635.321} C_VEL
LIN {X 0,Y 346.043,Z 761.494,A -85,B 0,C 180,E1 -13636.981,E2 -13636.981} C_VEL
LIN {X 0,Y 346.235,Z 759.757,A -85,B 0,C 180,E1 -13638.679,E2 -13638.679} C_VEL
LIN {X 0,Y 346.538,Z 757.065,A -85,B 0,C 180,E1 -13640.412,E2 -13640.412} C_VEL
LIN {X 0,Y 346.998,Z 753.302,A -85,B 0,C 180,E1 -13642.174,E2 -13642.174} C_VEL
LIN {X 0,Y 347.633,Z 747.876,A -85,B 0,C 180,E1 -13644.106,E2 -13644.106} C_VEL
LIN {X 0,Y 348.619,Z 740.458,A -85,B 0,C 180,E1 -13646.117,E2 -13646.117} C_VEL
LIN {X 0,Y 349.733,Z 732.384,A -85,B 0,C 180,E1 -13647.852,E2 -13647.852} C_VEL
LIN {X 0,Y 350.915,Z 723.067,A -85,B 0,C 180,E1 -13649.449,E2 -13649.449} C_VEL
LIN {X 0,Y 352.225,Z 712.65,A -85,B 0,C 180,E1 -13650.884,E2 -13650.884} C_VEL
LIN {X 0,Y 353.295,Z 702.957,A -85,B 0,C 180,E1 -13651.968,E2 -13651.968} C_VEL
LIN {X 0,Y 354.415,Z 691.21,A -85,B 0,C 180,E1 -13653.009,E2 -13653.009} C_VEL
LIN {X 0,Y 352.604,Z 679.586,A -85,B 0,C 180,E1 -13653.992,E2 -13653.992} C_VEL
LIN {X 0,Y 349.646,Z 667.458,A -85,B 0,C 180,E1 -13654.873,E2 -13654.873} C_VEL
LIN {X 0,Y 346.852,Z 658.013,A -85,B 0,C 180,E1 -13655.462,E2 -13655.462} C_VEL
LIN {X 0,Y 346.966,Z 653.439,A -85,B 0,C 180,E1 -13658.708,E2 -13658.708} C_VEL
LIN {X 0,Y 347.206,Z 648.251,A -85,B 0,C 180,E1 -13662.324,E2 -13662.324} C_VEL
LIN {X 0,Y 347.52,Z 642.813,A -85,B 0,C 180,E1 -13666.097,E2 -13666.097} C_VEL
LIN {X 0,Y 347.563,Z 641.199,A -85,B 0,C 180,E1 -13667.297,E2 -13667.297} C_VEL
LIN {X 0,Y 347.906,Z 641.152,A -85,B 0,C 180,E1 -13670.7,E2 -13670.7} C_VEL
LIN {X 0,Y 348.088,Z 641.13,A -85,B 0,C 180,E1 -13673.042,E2 -13673.042} C_VEL
LIN {X 0,Y 348.205,Z 641.113,A -85,B 0,C 180,E1 -13677.686,E2 -13677.686} C_VEL
LIN {X 0,Y 348.365,Z 641.094,A -85,B 0,C 180,E1 -13680,E2 -13680} C_VEL
LIN {X 0,Y 348.205,Z 641.113,A -85,B 0,C 180,E1 -13682.313,E2 -13682.313} C_VEL
LIN {X 0,Y 348.102,Z 641.125,A -85,B 0,C 180,E1 -13686.958,E2 -13686.958} C_VEL
LIN {X 0,Y 347.964,Z 641.142,A -85,B 0,C 180,E1 -13689.299,E2 -13689.299} C_VEL
LIN {X 0,Y 347.886,Z 641.153,A -85,B 0,C 180,E1 -13692.84,E2 -13692.84} C_VEL
LIN {X 0,Y 347.835,Z 641.157,A -85,B 0,C 180,E1 -13696.432,E2 -13696.432} C_VEL
LIN {X 0,Y 347.852,Z 641.154,A -85,B 0,C 180,E1 -13698.86,E2 -13698.86} C_VEL
LIN {X 0,Y 347.771,Z 641.167,A -85,B 0,C 180,E1 -13702.58,E2 -13702.58} C_VEL
LIN {X 0,Y 347.809,Z 641.162,A -85,B 0,C 180,E1 -13705.109,E2 -13705.109} C_VEL
LIN {X 0,Y 347.809,Z 641.162,A -85,B 0,C 180,E1 -13707.694,E2 -13707.694} C_VEL
LIN {X 0,Y 347.761,Z 641.167,A -85,B 0,C 180,E1 -13710.347,E2 -13710.347} C_VEL
LIN {X 0,Y 347.741,Z 641.171,A -85,B 0,C 180,E1 -13714.464,E2 -13714.464} C_VEL
LIN {X 0,Y 347.772,Z 641.164,A -85,B 0,C 180,E1 -13717.989,E2 -13717.989} C_VEL
LIN {X 0,Y 347.748,Z 641.167,A -85,B 0,C 180,E1 -13721.831,E2 -13721.831} C_VEL
LIN {X 0,Y 347.703,Z 641.176,A -85,B 0,C 180,E1 -13725.027,E2 -13725.027} C_VEL
LIN {X 0,Y 347.77,Z 641.245,A -85,B 0,C 180,E1 -13727.062,E2 -13727.062} C_VEL
LIN {X 0,Y 348.513,Z 645.36,A -85,B 0,C 180,E1 -13730.023,E2 -13730.023} C_VEL
LIN {X 0,Y 349.091,Z 649.464,A -85,B 0,C 180,E1 -13732.846,E2 -13732.846} C_VEL
LIN {X 0,Y 349.075,Z 653.762,A -85,B 0,C 180,E1 -13735.636,E2 -13735.636} C_VEL
LIN {X 0,Y 348.488,Z 659.277,A -85,B 0,C 180,E1 -13739.053,E2 -13739.053} C_VEL
LIN {X 0,Y 347.885,Z 665.396,A -85,B 0,C 180,E1 -13742.735,E2 -13742.735} C_VEL
LIN {X 0,Y 347.4,Z 671.169,A -85,B 0,C 180,E1 -13746.134,E2 -13746.134} C_VEL
LIN {X 0,Y 347.107,Z 676.142,A -85,B 0,C 180,E1 -13748.899,E2 -13748.899} C_VEL
LIN {X 0,Y 350.087,Z 689.593,A -85,B 0,C 180,E1 -13749.655,E2 -13749.655} C_VEL
LIN {X 0,Y 351.866,Z 702.331,A -85,B 0,C 180,E1 -13750.545,E2 -13750.545} C_VEL
LIN {X 0,Y 352.942,Z 714.298,A -85,B 0,C 180,E1 -13751.573,E2 -13751.573} C_VEL
LIN {X 0,Y 351.773,Z 726.054,A -85,B 0,C 180,E1 -13752.712,E2 -13752.712} C_VEL
LIN {X 0,Y 350.512,Z 736.989,A -85,B 0,C 180,E1 -13754.057,E2 -13754.057} C_VEL
LIN {X 0,Y 349.431,Z 746.084,A -85,B 0,C 180,E1 -13755.44,E2 -13755.44} C_VEL
LIN {X 0,Y 348.359,Z 755.279,A -85,B 0,C 180,E1 -13757.179,E2 -13757.179} C_VEL
LIN {X 0,Y 347.451,Z 762.638,A -85,B 0,C 180,E1 -13758.922,E2 -13758.922} C_VEL
LIN {X 0,Y 346.875,Z 768.779,A -85,B 0,C 180,E1 -13760.672,E2 -13760.672} C_VEL
LIN {X 0,Y 346.467,Z 773.781,A -85,B 0,C 180,E1 -13762.424,E2 -13762.424} C_VEL
LIN {X 0,Y 346.249,Z 777.635,A -85,B 0,C 180,E1 -13764.176,E2 -13764.176} C_VEL
LIN {X 0,Y 346.204,Z 779.616,A -85,B 0,C 180,E1 -13765.343,E2 -13765.343} C_VEL
LIN {X 0,Y 346.147,Z 781.175,A -85,B 0,C 180,E1 -13766.508,E2 -13766.508} C_VEL
LIN {X 0,Y 346.083,Z 782.284,A -85,B 0,C 180,E1 -13767.673,E2 -13767.673} C_VEL
LIN {X 0,Y 346.118,Z 782.972,A -85,B 0,C 180,E1 -13768.837,E2 -13768.837} C_VEL
LIN {X 0,Y 346.166,Z 783.267,A -85,B 0,C 180,E1 -13770,E2 -13770} C_VEL
LIN {X 0,Y 346.115,Z 783.166,A -85,B 0,C 180,E1 -13771.164,E2 -13771.164} C_VEL
LIN {X 0,Y 346.081,Z 782.637,A -85,B 0,C 180,E1 -13772.328,E2 -13772.328} C_VEL
LIN {X 0,Y 346.147,Z 781.692,A -85,B 0,C 180,E1 -13773.493,E2 -13773.493} C_VEL
LIN {X 0,Y 346.188,Z 780.347,A -85,B 0,C 180,E1 -13774.658,E2 -13774.658} C_VEL
LIN {X 0,Y 346.308,Z 777.521,A -85,B 0,C 180,E1 -13776.408,E2 -13776.408} C_VEL
LIN {X 0,Y 346.605,Z 773.668,A -85,B 0,C 180,E1 -13778.16,E2 -13778.16} C_VEL
LIN {X 0,Y 347.067,Z 768.694,A -85,B 0,C 180,E1 -13779.912,E2 -13779.912} C_VEL
LIN {X 0,Y 347.75,Z 762.456,A -85,B 0,C 180,E1 -13781.66,E2 -13781.66} C_VEL
LIN {X 0,Y 348.819,Z 754.719,A -85,B 0,C 180,E1 -13783.398,E2 -13783.398} C_VEL
LIN {X 0,Y 349.867,Z 746.832,A -85,B 0,C 180,E1 -13784.84,E2 -13784.84} C_VEL
LIN {X 0,Y 350.928,Z 737.259,A -85,B 0,C 180,E1 -13786.283,E2 -13786.283} C_VEL
LIN {X 0,Y 352.199,Z 726.709,A -85,B 0,C 180,E1 -13787.567,E2 -13787.567} C_VEL
LIN {X 0,Y 353.468,Z 715.354,A -85,B 0,C 180,E1 -13788.671,E2 -13788.671} C_VEL
LIN {X 0,Y 352.645,Z 703.631,A -85,B 0,C 180,E1 -13789.679,E2 -13789.679} C_VEL
LIN {X 0,Y 350.721,Z 691.515,A -85,B 0,C 180,E1 -13790.567,E2 -13790.567} C_VEL
LIN {X 0,Y 347.928,Z 679.162,A -85,B 0,C 180,E1 -13791.321,E2 -13791.321} C_VEL
LIN {X 0,Y 347.194,Z 675.986,A -85,B 0,C 180,E1 -13791.509,E2 -13791.509} C_VEL
LIN {X 0,Y 347.641,Z 669.905,A -85,B 0,C 180,E1 -13795.122,E2 -13795.122} C_VEL
LIN {X 0,Y 348.175,Z 664.699,A -85,B 0,C 180,E1 -13798.318,E2 -13798.318} C_VEL
LIN {X 0,Y 348.857,Z 658.66,A -85,B 0,C 180,E1 -13802.207,E2 -13802.207} C_VEL
LIN {X 0,Y 349.256,Z 655.382,A -85,B 0,C 180,E1 -13804.408,E2 -13804.408} C_VEL
LIN {X 0,Y 349.287,Z 651.599,A -85,B 0,C 180,E1 -13807.131,E2 -13807.131} C_VEL
LIN {X 0,Y 348.874,Z 647.787,A -85,B 0,C 180,E1 -13810.139,E2 -13810.139} C_VEL
LIN {X 0,Y 348.282,Z 644.026,A -85,B 0,C 180,E1 -13813.411,E2 -13813.411} C_VEL
LIN {X 0,Y 347.737,Z 641.173,A -85,B 0,C 180,E1 -13816.194,E2 -13816.194} C_VEL
LIN {X 0,Y 347.734,Z 641.175,A -85,B 0,C 180,E1 -13819.703,E2 -13819.703} C_VEL
LIN {X 0,Y 347.763,Z 641.168,A -85,B 0,C 180,E1 -13822.679,E2 -13822.679} C_VEL
LIN {X 0,Y 347.75,Z 641.168,A -85,B 0,C 180,E1 -13825.956,E2 -13825.956} C_VEL
LIN {X 0,Y 347.751,Z 641.167,A -85,B 0,C 180,E1 -13829.652,E2 -13829.652} C_VEL
LIN {X 0,Y 347.832,Z 641.156,A -85,B 0,C 180,E1 -13833.608,E2 -13833.608} C_VEL
LIN {X 0,Y 347.79,Z 641.16,A -85,B 0,C 180,E1 -13836.162,E2 -13836.162} C_VEL
LIN {X 0,Y 347.819,Z 641.16,A -85,B 0,C 180,E1 -13839.91,E2 -13839.91} C_VEL
LIN {X 0,Y 347.868,Z 641.155,A -85,B 0,C 180,E1 -13842.359,E2 -13842.359} C_VEL
LIN {X 0,Y 347.899,Z 641.15,A -85,B 0,C 180,E1 -13845.971,E2 -13845.971} C_VEL
LIN {X 0,Y 347.93,Z 641.146,A -85,B 0,C 180,E1 -13849.526,E2 -13849.526} C_VEL
LIN {X 0,Y 348.076,Z 641.126,A -85,B 0,C 180,E1 -13851.875,E2 -13851.875} C_VEL
LIN {X 0,Y 348.069,Z 641.127,A -85,B 0,C 180,E1 -13854.206,E2 -13854.206} C_VEL
LIN {X 0,Y 348.208,Z 641.111,A -85,B 0,C 180,E1 -13857.687,E2 -13857.687} C_VEL
LIN {X 0,Y 348.348,Z 641.095,A -85,B 0,C 180,E1 -13860,E2 -13860} C_VEL
LIN {X 0,Y 348.21,Z 641.115,A -85,B 0,C 180,E1 -13862.314,E2 -13862.314} C_VEL
LIN {X 0,Y 347.885,Z 641.154,A -85,B 0,C 180,E1 -13864.635,E2 -13864.635} C_VEL
LIN {X 0,Y 348.11,Z 641.544,A -85,B 0,C 180,E1 -13865.794,E2 -13865.794} C_VEL
LIN {X 0,Y 348.323,Z 643.998,A -85,B 0,C 180,E1 -13868.638,E2 -13868.638} C_VEL
LIN {X 0,Y 348.04,Z 646.838,A -85,B 0,C 180,E1 -13871.65,E2 -13871.65} C_VEL
LIN {X 0,Y 347.642,Z 650.408,A -85,B 0,C 180,E1 -13875.237,E2 -13875.237} C_VEL
LIN {X 0,Y 347.428,Z 653.327,A -85,B 0,C 180,E1 -13878.057,E2 -13878.057} C_VEL
LIN {X 0,Y 347.123,Z 656.904,A -85,B 0,C 180,E1 -13881.373,E2 -13881.373} C_VEL
LIN {X 0,Y 346.976,Z 659.342,A -85,B 0,C 180,E1 -13883.581,E2 -13883.581} C_VEL
LIN {X 0,Y 351.139,Z 673.437,A -85,B 0,C 180,E1 -13884.527,E2 -13884.527} C_VEL
LIN {X 0,Y 353.613,Z 684.939,A -85,B 0,C 180,E1 -13885.435,E2 -13885.435} C_VEL
LIN {X 0,Y 354.621,Z 691.586,A -85,B 0,C 180,E1 -13886.023,E2 -13886.023} C_VEL
LIN {X 0,Y 353.406,Z 703.221,A -85,B 0,C 180,E1 -13887.061,E2 -13887.061} C_VEL
LIN {X 0,Y 352.271,Z 713.597,A -85,B 0,C 180,E1 -13888.233,E2 -13888.233} C_VEL
LIN {X 0,Y 351.02,Z 723.078,A -85,B 0,C 180,E1 -13889.54,E2 -13889.54} C_VEL
LIN {X 0,Y 349.972,Z 731.158,A -85,B 0,C 180,E1 -13890.901,E2 -13890.901} C_VEL
LIN {X 0,Y 348.926,Z 739.249,A -85,B 0,C 180,E1 -13892.568,E2 -13892.568} C_VEL
LIN {X 0,Y 347.922,Z 746.497,A -85,B 0,C 180,E1 -13894.444,E2 -13894.444} C_VEL
LIN {X 0,Y 347.334,Z 751.215,A -85,B 0,C 180,E1 -13895.966,E2 -13895.966} C_VEL
LIN {X 0,Y 346.784,Z 755.659,A -85,B 0,C 180,E1 -13897.778,E2 -13897.778} C_VEL
LIN {X 0,Y 346.435,Z 758.92,A -85,B 0,C 180,E1 -13899.566,E2 -13899.566} C_VEL
LIN {X 0,Y 346.161,Z 761.118,A -85,B 0,C 180,E1 -13901.305,E2 -13901.305} C_VEL
LIN {X 0,Y 345.963,Z 762.653,A -85,B 0,C 180,E1 -13903.685,E2 -13903.685} C_VEL
LIN {X 0,Y 345.92,Z 762.713,A -85,B 0,C 180,E1 -13905.324,E2 -13905.324} C_VEL
LIN {X 0,Y 345.994,Z 761.973,A -85,B 0,C 180,E1 -13906.992,E2 -13906.992} C_VEL
LIN {X 0,Y 346.139,Z 760.362,A -85,B 0,C 180,E1 -13908.699,E2 -13908.699} C_VEL
LIN {X 0,Y 346.413,Z 757.787,A -85,B 0,C 180,E1 -13910.439,E2 -13910.439} C_VEL
LIN {X 0,Y 346.744,Z 753.292,A -85,B 0,C 180,E1 -13912.551,E2 -13912.551} C_VEL
LIN {X 0,Y 347.292,Z 747.877,A -85,B 0,C 180,E1 -13914.442,E2 -13914.442} C_VEL
LIN {X 0,Y 347.963,Z 741.46,A -85,B 0,C 180,E1 -13916.203,E2 -13916.203} C_VEL
LIN {X 0,Y 348.773,Z 734.143,A -85,B 0,C 180,E1 -13917.815,E2 -13917.815} C_VEL
LIN {X 0,Y 349.758,Z 724.916,A -85,B 0,C 180,E1 -13919.462,E2 -13919.462} C_VEL
LIN {X 0,Y 350.954,Z 714.56,A -85,B 0,C 180,E1 -13920.947,E2 -13920.947} C_VEL
LIN {X 0,Y 351.981,Z 703.797,A -85,B 0,C 180,E1 -13922.177,E2 -13922.177} C_VEL
LIN {X 0,Y 352.954,Z 692.3,A -85,B 0,C 180,E1 -13923.224,E2 -13923.224} C_VEL
LIN {X 0,Y 353.063,Z 688.707,A -85,B 0,C 180,E1 -13923.508,E2 -13923.508} C_VEL
LIN {X 0,Y 350.77,Z 675.92,A -85,B 0,C 180,E1 -13924.483,E2 -13924.483} C_VEL
LIN {X 0,Y 347.872,Z 663.102,A -85,B 0,C 180,E1 -13925.244,E2 -13925.244} C_VEL
LIN {X 0,Y 346.688,Z 658.209,A -85,B 0,C 180,E1 -13925.51,E2 -13925.51} C_VEL
LIN {X 0,Y 346.862,Z 654.324,A -85,B 0,C 180,E1 -13928.755,E2 -13928.755} C_VEL
LIN {X 0,Y 347.145,Z 650.148,A -85,B 0,C 180,E1 -13932.321,E2 -13932.321} C_VEL
LIN {X 0,Y 347.476,Z 645.787,A -85,B 0,C 180,E1 -13936.131,E2 -13936.131} C_VEL
LIN {X 0,Y 347.692,Z 642.032,A -85,B 0,C 180,E1 -13939.518,E2 -13939.518} C_VEL
LIN {X 0,Y 347.735,Z 641.383,A -85,B 0,C 180,E1 -13940.108,E2 -13940.108} C_VEL
LIN {X 0,Y 348.026,Z 641.13,A -85,B 0,C 180,E1 -13941.873,E2 -13941.873} C_VEL
LIN {X 0,Y 348.064,Z 641.126,A -85,B 0,C 180,E1 -13944.205,E2 -13944.205} C_VEL
LIN {X 0,Y 348.211,Z 641.107,A -85,B 0,C 180,E1 -13947.686,E2 -13947.686} C_VEL
LIN {X 0,Y 348.35,Z 641.09,A -85,B 0,C 180,E1 -13950,E2 -13950} C_VEL
LIN {X 0,Y 348.211,Z 641.108,A -85,B 0,C 180,E1 -13952.313,E2 -13952.313} C_VEL
LIN {X 0,Y 348.057,Z 641.131,A -85,B 0,C 180,E1 -13956.958,E2 -13956.958} C_VEL
LIN {X 0,Y 347.749,Z 641.166,A -85,B 0,C 180,E1 -13959.304,E2 -13959.304} C_VEL
LIN {X 0,Y 347.262,Z 641.227,A -85,B 0,C 180,E1 -13962.268,E2 -13962.268} C_VEL
LIN {X 0,Y 346.892,Z 647.18,A -85,B 0,C 180,E1 -13966.477,E2 -13966.477} C_VEL
LIN {X 0,Y 346.756,Z 650.636,A -85,B 0,C 180,E1 -13968.922,E2 -13968.922} C_VEL
LIN {X 0,Y 346.582,Z 655.914,A -85,B 0,C 180,E1 -13972.661,E2 -13972.661} C_VEL
LIN {X 0,Y 346.562,Z 657.277,A -85,B 0,C 180,E1 -13973.61,E2 -13973.61} C_VEL
LIN {X 0,Y 350.003,Z 672.17,A -85,B 0,C 180,E1 -13974.423,E2 -13974.423} C_VEL
LIN {X 0,Y 352.54,Z 685.535,A -85,B 0,C 180,E1 -13975.379,E2 -13975.379} C_VEL
LIN {X 0,Y 353.05,Z 689.879,A -85,B 0,C 180,E1 -13975.734,E2 -13975.734} C_VEL
LIN {X 0,Y 352.051,Z 701.736,A -85,B 0,C 180,E1 -13976.759,E2 -13976.759} C_VEL
LIN {X 0,Y 351,Z 712.625,A -85,B 0,C 180,E1 -13977.964,E2 -13977.964} C_VEL
LIN {X 0,Y 349.856,Z 723.565,A -85,B 0,C 180,E1 -13979.482,E2 -13979.482} C_VEL
LIN {X 0,Y 348.918,Z 731.869,A -85,B 0,C 180,E1 -13980.905,E2 -13980.905} C_VEL
LIN {X 0,Y 348.062,Z 739.532,A -85,B 0,C 180,E1 -13982.517,E2 -13982.517} C_VEL
LIN {X 0,Y 347.271,Z 747.113,A -85,B 0,C 180,E1 -13984.517,E2 -13984.517} C_VEL
LIN {X 0,Y 347.035,Z 749.782,A -85,B 0,C 180,E1 -13985.379,E2 -13985.379} C_VEL
LIN {X 0,Y 346.118,Z 752.311,A -85,B 0,C 180,E1 -13986.254,E2 -13986.254} C_VEL
LIN {X 0,Y 341.528,Z 757.119,A -85,B 0,C 180,E1 -13988.289,E2 -13988.289} C_VEL
LIN {X 0,Y 339.38,Z 759.188,A -85,B 0,C 180,E1 -13989.528,E2 -13989.528} C_VEL
LIN {X 0,Y 338.966,Z 759.987,A -85,B 0,C 180,E1 -13990.18,E2 -13990.18} C_VEL
LIN {X 0,Y 338.817,Z 761.572,A -85,B 0,C 180,E1 -13991.691,E2 -13991.691} C_VEL
LIN {X 0,Y 338.807,Z 762.529,A -85,B 0,C 180,E1 -13993.446,E2 -13993.446} C_VEL
LIN {X 0,Y 338.832,Z 762.6,A -85,B 0,C 180,E1 -13995.152,E2 -13995.152} C_VEL
LIN {X 0,Y 338.949,Z 761.87,A -85,B 0,C 180,E1 -13996.823,E2 -13996.823} C_VEL
LIN {X 0,Y 339.108,Z 760.398,A -85,B 0,C 180,E1 -13998.455,E2 -13998.455} C_VEL
LIN {X 0,Y 339.375,Z 758.197,A -85,B 0,C 180,E1 -14000.061,E2 -14000.061} C_VEL
LIN {X 0,Y 339.827,Z 754.881,A -85,B 0,C 180,E1 -14001.801,E2 -14001.801} C_VEL
LIN {X 0,Y 340.394,Z 750.265,A -85,B 0,C 180,E1 -14003.63,E2 -14003.63} C_VEL
LIN {X 0,Y 341.197,Z 744.267,A -85,B 0,C 180,E1 -14005.478,E2 -14005.478} C_VEL
LIN {X 0,Y 342.247,Z 736.657,A -85,B 0,C 180,E1 -14007.343,E2 -14007.343} C_VEL
LIN {X 0,Y 343.405,Z 728.843,A -85,B 0,C 180,E1 -14008.886,E2 -14008.886} C_VEL
LIN {X 0,Y 344.656,Z 719.63,A -85,B 0,C 180,E1 -14010.364,E2 -14010.364} C_VEL
LIN {X 0,Y 346.028,Z 708.353,A -85,B 0,C 180,E1 -14011.821,E2 -14011.821} C_VEL
LIN {X 0,Y 347.263,Z 697.428,A -85,B 0,C 180,E1 -14012.932,E2 -14012.932} C_VEL
LIN {X 0,Y 347.709,Z 691.769,A -85,B 0,C 180,E1 -14013.42,E2 -14013.42} C_VEL
LIN {X 0,Y 345.784,Z 680.165,A -85,B 0,C 180,E1 -14014.441,E2 -14014.441} C_VEL
LIN {X 0,Y 342.723,Z 667.719,A -85,B 0,C 180,E1 -14015.384,E2 -14015.384} C_VEL
LIN {X 0,Y 339.818,Z 658.207,A -85,B 0,C 180,E1 -14016.013,E2 -14016.013} C_VEL
LIN {X 0,Y 339.948,Z 653.421,A -85,B 0,C 180,E1 -14019.424,E2 -14019.424} C_VEL
LIN {X 0,Y 340.141,Z 649.905,A -85,B 0,C 180,E1 -14021.945,E2 -14021.945} C_VEL
LIN {X 0,Y 340.476,Z 644.163,A -85,B 0,C 180,E1 -14025.964,E2 -14025.964} C_VEL
LIN {X 0,Y 340.534,Z 642.074,A -85,B 0,C 180,E1 -14027.485,E2 -14027.485} C_VEL
LIN {X 0,Y 340.843,Z 642.031,A -85,B 0,C 180,E1 -14030.505,E2 -14030.505} C_VEL
LIN {X 0,Y 341.055,Z 642.006,A -85,B 0,C 180,E1 -14032.898,E2 -14032.898} C_VEL
LIN {X 0,Y 341.167,Z 641.989,A -85,B 0,C 180,E1 -14037.639,E2 -14037.639} C_VEL
LIN {X 0,Y 341.314,Z 641.972,A -85,B 0,C 180,E1 -14040,E2 -14040} C_VEL
LIN {X 0,Y 341.167,Z 641.99,A -85,B 0,C 180,E1 -14042.361,E2 -14042.361} C_VEL
LIN {X 0,Y 341.072,Z 642.001,A -85,B 0,C 180,E1 -14047.102,E2 -14047.102} C_VEL
LIN {X 0,Y 340.867,Z 642.028,A -85,B 0,C 180,E1 -14050.694,E2 -14050.694} C_VEL
LIN {X 0,Y 340.859,Z 642.025,A -85,B 0,C 180,E1 -14054.325,E2 -14054.325} C_VEL
LIN {X 0,Y 340.834,Z 642.03,A -85,B 0,C 180,E1 -14058.467,E2 -14058.467} C_VEL
LIN {X 0,Y 340.75,Z 642.039,A -85,B 0,C 180,E1 -14061.857,E2 -14061.857} C_VEL
LIN {X 0,Y 340.769,Z 642.038,A -85,B 0,C 180,E1 -14065.665,E2 -14065.665} C_VEL
LIN {X 0,Y 340.739,Z 642.04,A -85,B 0,C 180,E1 -14068.32,E2 -14068.32} C_VEL
LIN {X 0,Y 340.701,Z 642.045,A -85,B 0,C 180,E1 -14071.044,E2 -14071.044} C_VEL
LIN {X 0,Y 340.715,Z 642.044,A -85,B 0,C 180,E1 -14075.279,E2 -14075.279} C_VEL
LIN {X 0,Y 340.708,Z 642.046,A -85,B 0,C 180,E1 -14078.387,E2 -14078.387} C_VEL
LIN {X 0,Y 340.696,Z 642.045,A -85,B 0,C 180,E1 -14082.046,E2 -14082.046} C_VEL
LIN {X 0,Y 340.664,Z 642.052,A -85,B 0,C 180,E1 -14086.225,E2 -14086.225} C_VEL
LIN {X 0,Y 340.73,Z 642.217,A -85,B 0,C 180,E1 -14086.889,E2 -14086.889} C_VEL
LIN {X 0,Y 341.597,Z 646.972,A -85,B 0,C 180,E1 -14090.374,E2 -14090.374} C_VEL
LIN {X 0,Y 341.976,Z 649.184,A -85,B 0,C 180,E1 -14091.937,E2 -14091.937} C_VEL
LIN {X 0,Y 342.137,Z 653.567,A -85,B 0,C 180,E1 -14094.89,E2 -14094.89} C_VEL
LIN {X 0,Y 341.52,Z 659.002,A -85,B 0,C 180,E1 -14098.349,E2 -14098.349} C_VEL
LIN {X 0,Y 340.985,Z 664.416,A -85,B 0,C 180,E1 -14101.703,E2 -14101.703} C_VEL
LIN {X 0,Y 340.394,Z 670.89,A -85,B 0,C 180,E1 -14105.611,E2 -14105.611} C_VEL
LIN {X 0,Y 340.085,Z 675.623,A -85,B 0,C 180,E1 -14108.347,E2 -14108.347} C_VEL
LIN {X 0,Y 343.199,Z 689.25,A -85,B 0,C 180,E1 -14109.15,E2 -14109.15} C_VEL
LIN {X 0,Y 344.98,Z 701.369,A -85,B 0,C 180,E1 -14110.018,E2 -14110.018} C_VEL
LIN {X 0,Y 346.081,Z 713.106,A -85,B 0,C 180,E1 -14111.04,E2 -14111.04} C_VEL
LIN {X 0,Y 345.864,Z 719.446,A -85,B 0,C 180,E1 -14111.642,E2 -14111.642} C_VEL
LIN {X 0,Y 344.584,Z 730.07,A -85,B 0,C 180,E1 -14112.799,E2 -14112.799} C_VEL
LIN {X 0,Y 343.311,Z 740.24,A -85,B 0,C 180,E1 -14114.186,E2 -14114.186} C_VEL
LIN {X 0,Y 342.148,Z 749.429,A -85,B 0,C 180,E1 -14115.731,E2 -14115.731} C_VEL
LIN {X 0,Y 341.05,Z 757.912,A -85,B 0,C 180,E1 -14117.504,E2 -14117.504} C_VEL
LIN {X 0,Y 340.24,Z 764.74,A -85,B 0,C 180,E1 -14119.287,E2 -14119.287} C_VEL
LIN {X 0,Y 339.522,Z 771.913,A -85,B 0,C 180,E1 -14121.669,E2 -14121.669} C_VEL
LIN {X 0,Y 339.227,Z 776.163,A -85,B 0,C 180,E1 -14123.458,E2 -14123.458} C_VEL
LIN {X 0,Y 339.105,Z 779.334,A -85,B 0,C 180,E1 -14125.245,E2 -14125.245} C_VEL
LIN {X 0,Y 339.073,Z 780.906,A -85,B 0,C 180,E1 -14126.436,E2 -14126.436} C_VEL
LIN {X 0,Y 338.998,Z 782.041,A -85,B 0,C 180,E1 -14127.624,E2 -14127.624} C_VEL
LIN {X 0,Y 339.02,Z 782.74,A -85,B 0,C 180,E1 -14128.813,E2 -14128.813} C_VEL
LIN {X 0,Y 339.069,Z 783.047,A -85,B 0,C 180,E1 -14130.001,E2 -14130.001} C_VEL
LIN {X 0,Y 339.017,Z 782.959,A -85,B 0,C 180,E1 -14131.188,E2 -14131.188} C_VEL
LIN {X 0,Y 338.996,Z 782.456,A -85,B 0,C 180,E1 -14132.377,E2 -14132.377} C_VEL
LIN {X 0,Y 339.072,Z 781.525,A -85,B 0,C 180,E1 -14133.566,E2 -14133.566} C_VEL
LIN {X 0,Y 339.091,Z 780.194,A -85,B 0,C 180,E1 -14134.756,E2 -14134.756} C_VEL
LIN {X 0,Y 339.243,Z 777.394,A -85,B 0,C 180,E1 -14136.543,E2 -14136.543} C_VEL
LIN {X 0,Y 339.555,Z 773.568,A -85,B 0,C 180,E1 -14138.331,E2 -14138.331} C_VEL
LIN {X 0,Y 340.059,Z 768.623,A -85,B 0,C 180,E1 -14140.118,E2 -14140.118} C_VEL
LIN {X 0,Y 340.776,Z 762.416,A -85,B 0,C 180,E1 -14141.902,E2 -14141.902} C_VEL
LIN {X 0,Y 341.908,Z 754.728,A -85,B 0,C 180,E1 -14143.674,E2 -14143.674} C_VEL
LIN {X 0,Y 342.976,Z 746.911,A -85,B 0,C 180,E1 -14145.145,E2 -14145.145} C_VEL
LIN {X 0,Y 344.116,Z 737.43,A -85,B 0,C 180,E1 -14146.615,E2 -14146.615} C_VEL
LIN {X 0,Y 345.464,Z 726.993,A -85,B 0,C 180,E1 -14147.921,E2 -14147.921} C_VEL
LIN {X 0,Y 346.741,Z 715.815,A -85,B 0,C 180,E1 -14149.045,E2 -14149.045} C_VEL
LIN {X 0,Y 345.914,Z 704.318,A -85,B 0,C 180,E1 -14150.078,E2 -14150.078} C_VEL
LIN {X 0,Y 343.988,Z 691.971,A -85,B 0,C 180,E1 -14151.019,E2 -14151.019} C_VEL
LIN {X 0,Y 340.915,Z 678.696,A -85,B 0,C 180,E1 -14151.874,E2 -14151.874} C_VEL
LIN {X 0,Y 340.231,Z 675.767,A -85,B 0,C 180,E1 -14152.043,E2 -14152.043} C_VEL
LIN {X 0,Y 340.681,Z 669.835,A -85,B 0,C 180,E1 -14155.672,E2 -14155.672} C_VEL
LIN {X 0,Y 341.198,Z 664.667,A -85,B 0,C 180,E1 -14158.951,E2 -14158.951} C_VEL
LIN {X 0,Y 341.909,Z 659.214,A -85,B 0,C 180,E1 -14162.567,E2 -14162.567} C_VEL
LIN {X 0,Y 342.292,Z 655.599,A -85,B 0,C 180,E1 -14165.093,E2 -14165.093} C_VEL
LIN {X 0,Y 342.335,Z 653.274,A -85,B 0,C 180,E1 -14166.807,E2 -14166.807} C_VEL
LIN {X 0,Y 341.993,Z 649.798,A -85,B 0,C 180,E1 -14169.573,E2 -14169.573} C_VEL
LIN {X 0,Y 341.418,Z 646.123,A -85,B 0,C 180,E1 -14172.789,E2 -14172.789} C_VEL
LIN {X 0,Y 340.716,Z 642.201,A -85,B 0,C 180,E1 -14176.649,E2 -14176.649} C_VEL
LIN {X 0,Y 340.701,Z 642.049,A -85,B 0,C 180,E1 -14180.248,E2 -14180.248} C_VEL
LIN {X 0,Y 340.712,Z 642.047,A -85,B 0,C 180,E1 -14183.559,E2 -14183.559} C_VEL
LIN {X 0,Y 340.694,Z 642.047,A -85,B 0,C 180,E1 -14186.153,E2 -14186.153} C_VEL
LIN {X 0,Y 340.743,Z 642.042,A -85,B 0,C 180,E1 -14190.329,E2 -14190.329} C_VEL
LIN {X 0,Y 340.805,Z 642.035,A -85,B 0,C 180,E1 -14193.02,E2 -14193.02} C_VEL
LIN {X 0,Y 340.758,Z 642.037,A -85,B 0,C 180,E1 -14195.638,E2 -14195.638} C_VEL
LIN {X 0,Y 340.75,Z 642.042,A -85,B 0,C 180,E1 -14199.474,E2 -14199.474} C_VEL
LIN {X 0,Y 340.86,Z 642.028,A -85,B 0,C 180,E1 -14201.984,E2 -14201.984} C_VEL
LIN {X 0,Y 340.871,Z 642.027,A -85,B 0,C 180,E1 -14205.705,E2 -14205.705} C_VEL
LIN {X 0,Y 340.873,Z 642.027,A -85,B 0,C 180,E1 -14209.306,E2 -14209.306} C_VEL
LIN {X 0,Y 341.077,Z 642.001,A -85,B 0,C 180,E1 -14212.898,E2 -14212.898} C_VEL
LIN {X 0,Y 341.17,Z 641.988,A -85,B 0,C 180,E1 -14217.639,E2 -14217.639} C_VEL
LIN {X 0,Y 341.298,Z 641.973,A -85,B 0,C 180,E1 -14220,E2 -14220} C_VEL
LIN {X 0,Y 341.172,Z 641.991,A -85,B 0,C 180,E1 -14222.361,E2 -14222.361} C_VEL
LIN {X 0,Y 340.849,Z 642.03,A -85,B 0,C 180,E1 -14224.731,E2 -14224.731} C_VEL
LIN {X 0,Y 341.275,Z 643.859,A -85,B 0,C 180,E1 -14227.098,E2 -14227.098} C_VEL
LIN {X 0,Y 341.257,Z 645.945,A -85,B 0,C 180,E1 -14229.483,E2 -14229.483} C_VEL
LIN {X 0,Y 340.865,Z 649.353,A -85,B 0,C 180,E1 -14233.109,E2 -14233.109} C_VEL
LIN {X 0,Y 340.485,Z 653.018,A -85,B 0,C 180,E1 -14236.797,E2 -14236.797} C_VEL
LIN {X 0,Y 340.226,Z 655.611,A -85,B 0,C 180,E1 -14239.3,E2 -14239.3} C_VEL
LIN {X 0,Y 339.944,Z 659.564,A -85,B 0,C 180,E1 -14243.009,E2 -14243.009} C_VEL
LIN {X 0,Y 344.417,Z 674.51,A -85,B 0,C 180,E1 -14244.086,E2 -14244.086} C_VEL
LIN {X 0,Y 346.835,Z 685.387,A -85,B 0,C 180,E1 -14244.985,E2 -14244.985} C_VEL
LIN {X 0,Y 347.895,Z 693.656,A -85,B 0,C 180,E1 -14245.743,E2 -14245.743} C_VEL
LIN {X 0,Y 346.564,Z 705.322,A -85,B 0,C 180,E1 -14246.839,E2 -14246.839} C_VEL
LIN {X 0,Y 345.351,Z 715.505,A -85,B 0,C 180,E1 -14248.048,E2 -14248.048} C_VEL
LIN {X 0,Y 343.962,Z 725.558,A -85,B 0,C 180,E1 -14249.534,E2 -14249.534} C_VEL
LIN {X 0,Y 342.702,Z 734.553,A -85,B 0,C 180,E1 -14251.186,E2 -14251.186} C_VEL
LIN {X 0,Y 341.704,Z 741.643,A -85,B 0,C 180,E1 -14252.79,E2 -14252.79} C_VEL
LIN {X 0,Y 340.859,Z 747.595,A -85,B 0,C 180,E1 -14254.438,E2 -14254.438} C_VEL
LIN {X 0,Y 340.137,Z 752.988,A -85,B 0,C 180,E1 -14256.309,E2 -14256.309} C_VEL
LIN {X 0,Y 339.599,Z 757.444,A -85,B 0,C 180,E1 -14258.378,E2 -14258.378} C_VEL
LIN {X 0,Y 339.269,Z 759.96,A -85,B 0,C 180,E1 -14259.963,E2 -14259.963} C_VEL
LIN {X 0,Y 339.039,Z 761.849,A -85,B 0,C 180,E1 -14261.733,E2 -14261.733} C_VEL
LIN {X 0,Y 338.894,Z 762.813,A -85,B 0,C 180,E1 -14263.462,E2 -14263.462} C_VEL
LIN {X 0,Y 338.838,Z 762.946,A -85,B 0,C 180,E1 -14265.153,E2 -14265.153} C_VEL
LIN {X 0,Y 338.902,Z 762.3,A -85,B 0,C 180,E1 -14266.816,E2 -14266.816} C_VEL
LIN {X 0,Y 339.024,Z 760.911,A -85,B 0,C 180,E1 -14268.443,E2 -14268.443} C_VEL
LIN {X 0,Y 339.373,Z 757.396,A -85,B 0,C 180,E1 -14270.83,E2 -14270.83} C_VEL
LIN {X 0,Y 339.636,Z 753.861,A -85,B 0,C 180,E1 -14272.506,E2 -14272.506} C_VEL
LIN {X 0,Y 340.095,Z 749.292,A -85,B 0,C 180,E1 -14274.193,E2 -14274.193} C_VEL
LIN {X 0,Y 340.835,Z 742.484,A -85,B 0,C 180,E1 -14276.169,E2 -14276.169} C_VEL
LIN {X 0,Y 341.818,Z 734.305,A -85,B 0,C 180,E1 -14278.032,E2 -14278.032} C_VEL
LIN {X 0,Y 342.786,Z 725.357,A -85,B 0,C 180,E1 -14279.665,E2 -14279.665} C_VEL
